    movel([0.098799, -1.267292, -2.641925, -0.803171, 1.570796, 1.669595],accel_mss,speed_ms,0,blend_radius_m)
    movel([0.098967, -1.267010, -2.642082, -0.803297, 1.570796, 1.669764],accel_mss,speed_ms,0,blend_radius_m)
    movel([0.099464, -1.266678, -2.642266, -0.803445, 1.570796, 1.670261],accel_mss,speed_ms,0,blend_radius_m)
    speed_ms = 0.003
    movel([0.099464, -1.270243, -2.643943, -0.798203, 1.570796, 1.670261],accel_mss,speed_ms,0,blend_radius_m)
    speed_ms = 0.007
    movel([0.099864, -1.269963, -2.644099, -0.798327, 1.570796, 1.670661],accel_mss,speed_ms,0,blend_radius_m)
    movel([0.100140, -1.269497, -2.644358, -0.798534, 1.570796, 1.670936],accel_mss,speed_ms,0,blend_radius_m)
    movel([0.100356, -1.268649, -2.644829, -0.798911, 1.570796, 1.671153],accel_mss,speed_ms,0,blend_radius_m)
    movel([0.100640, -1.266818, -2.645843, -0.799728, 1.570796, 1.671436],accel_mss,speed_ms,0,blend_radius_m)
    movel([0.100880, -1.265181, -2.646746, -0.800463, 1.570796, 1.671677],accel_mss,speed_ms,0,blend_radius_m)
    movel([0.101009, -1.264534, -2.647102, -0.800754, 1.570796, 1.671805],accel_mss,speed_ms,0,blend_radius_m)
    movel([0.101145, -1.264159, -2.647307, -0.800923, 1.570796, 1.671942],accel_mss,speed_ms,0,blend_radius_m)
    movel([0.101358, -1.263870, -2.647466, -0.801053, 1.570796, 1.672154],accel_mss,speed_ms,0,blend_radius_m)
    movel([0.101658, -1.263620, -2.647603, -0.801166, 1.570796, 1.672454],accel_mss,speed_ms,0,blend_radius_m)
    movel([0.102128, -1.263533, -2.647651, -0.801205, 1.570796, 1.672924],accel_mss,speed_ms,0,blend_radius_m)
    movel([0.102340, -1.263694, -2.647563, -0.801132, 1.570796, 1.673136],accel_mss,speed_ms,0,blend_radius_m)
    movel([0.102446, -1.263926, -2.647435, -0.801028, 1.570796, 1.673242],accel_mss,speed_ms,0,blend_radius_m)
    movel([0.102458, -1.264305, -2.647228, -0.800857, 1.570796, 1.673254],accel_mss,speed_ms,0,blend_radius_m)
    movel([0.102379, -1.264992, -2.646850, -0.800548, 1.570796, 1.673176],accel_mss,speed_ms,0,blend_radius_m)
    movel([0.102123, -1.266603, -2.645961, -0.799825, 1.570796, 1.672919],accel_mss,speed_ms,0,blend_radius_m)
    movel([0.101853, -1.268341, -2.645000, -0.799048, 1.570796, 1.672649],accel_mss,speed_ms,0,blend_radius_m)
    movel([0.101798, -1.269088, -2.644586, -0.798716, 1.570796, 1.672594],accel_mss,speed_ms,0,blend_radius_m)
    movel([0.101884, -1.269413, -2.644405, -0.798571, 1.570796, 1.672681],accel_mss,speed_ms,0,blend_radius_m)
    movel([0.102127, -1.269459, -2.644379, -0.798551, 1.570796, 1.672923],accel_mss,speed_ms,0,blend_radius_m)
    movel([0.102418, -1.269491, -2.644362, -0.798537, 1.570796, 1.673214],accel_mss,speed_ms,0,blend_radius_m)
    movel([0.102637, -1.269624, -2.644288, -0.798478, 1.570796, 1.673433],accel_mss,speed_ms,0,blend_radius_m)
    movel([0.102685, -1.269900, -2.644134, -0.798355, 1.570796, 1.673481],accel_mss,speed_ms,0,blend_radius_m)
    movel([0.102479, -1.270544, -2.643776, -0.798070, 1.570796, 1.673275],accel_mss,speed_ms,0,blend_radius_m)
    movel([0.102314, -1.270823, -2.643620, -0.797946, 1.570796, 1.673111],accel_mss,speed_ms,0,blend_radius_m)
    movel([0.101871, -1.271146, -2.643440, -0.797803, 1.570796, 1.672667],accel_mss,speed_ms,0,blend_radius_m)
    movel([0.101580, -1.271362, -2.643319, -0.797707, 1.570796, 1.672376],accel_mss,speed_ms,0,blend_radius_m)
    movel([0.101261, -1.271773, -2.643090, -0.797526, 1.570796, 1.672057],accel_mss,speed_ms,0,blend_radius_m)
    movel([0.100848, -1.272313, -2.642788, -0.797288, 1.570796, 1.671644],accel_mss,speed_ms,0,blend_radius_m)
    movel([0.100469, -1.272559, -2.642650, -0.797179, 1.570796, 1.671265],accel_mss,speed_ms,0,blend_radius_m)
    movel([0.100136, -1.272520, -2.642672, -0.797197, 1.570796, 1.670932],accel_mss,speed_ms,0,blend_radius_m)
    movel([0.099864, -1.272178, -2.642863, -0.797347, 1.570796, 1.670660],accel_mss,speed_ms,0,blend_radius_m)
    movel([0.099641, -1.271932, -2.643001, -0.797456, 1.570796, 1.670438],accel_mss,speed_ms,0,blend_radius_m)
    movel([0.099334, -1.271905, -2.643016, -0.797468, 1.570796, 1.670130],accel_mss,speed_ms,0,blend_radius_m)
    movel([0.098951, -1.271937, -2.642998, -0.797454, 1.570796, 1.669747],accel_mss,speed_ms,0,blend_radius_m)
    movel([0.098703, -1.271840, -2.643053, -0.797497, 1.570796, 1.669500],accel_mss,speed_ms,0,blend_radius_m)
    movel([0.098605, -1.271610, -2.643181, -0.797598, 1.570796, 1.669401],accel_mss,speed_ms,0,blend_radius_m)
    movel([0.098652, -1.271263, -2.643375, -0.797751, 1.570796, 1.669448],accel_mss,speed_ms,0,blend_radius_m)
    movel([0.098799, -1.270856, -2.643602, -0.797931, 1.570796, 1.669595],accel_mss,speed_ms,0,blend_radius_m)
    movel([0.098967, -1.270575, -2.643758, -0.798056, 1.570796, 1.669764],accel_mss,speed_ms,0,blend_radius_m)
    movel([0.099464, -1.270243, -2.643943, -0.798203, 1.570796, 1.670261],accel_mss,speed_ms,0,blend_radius_m)
    speed_ms = 0.003
    movel([0.099464, -1.256163, -2.637185, -0.819041, 1.570796, 1.670261],accel_mss,speed_ms,0,blend_radius_m)
    speed_ms = 1.000
    movel([0.099464, -1.229425, -2.623288, -0.859676, 1.570796, 1.670261],accel_mss,speed_ms,0,blend_radius_m)
    movel([0.085805, -1.233581, -2.621092, -0.857716, 1.570796, 1.656601],accel_mss,speed_ms,0,blend_radius_m)
    movel([0.085805, -1.260270, -2.634934, -0.817185, 1.570796, 1.656601],accel_mss,speed_ms,0,blend_radius_m)
    speed_ms = 0.003
    movel([0.085805, -1.270762, -2.639994, -0.801634, 1.570796, 1.656601],accel_mss,speed_ms,0,blend_radius_m)
    speed_ms = 0.007
    movel([0.086070, -1.265880, -2.642708, -0.803802, 1.570796, 1.656867],accel_mss,speed_ms,0,blend_radius_m)
    movel([0.086295, -1.263990, -2.643750, -0.804649, 1.570796, 1.657092],accel_mss,speed_ms,0,blend_radius_m)
    movel([0.086599, -1.262035, -2.644825, -0.805530, 1.570796, 1.657396],accel_mss,speed_ms,0,blend_radius_m)
    movel([0.086929, -1.260286, -2.645781, -0.806321, 1.570796, 1.657725],accel_mss,speed_ms,0,blend_radius_m)
    movel([0.087180, -1.259543, -2.646187, -0.806659, 1.570796, 1.657976],accel_mss,speed_ms,0,blend_radius_m)
    movel([0.087885, -1.258813, -2.646585, -0.806992, 1.570796, 1.658681],accel_mss,speed_ms,0,blend_radius_m)
    movel([0.089726, -1.257950, -2.647054, -0.807385, 1.570796, 1.660522],accel_mss,speed_ms,0,blend_radius_m)
    movel([0.092956, -1.256741, -2.647709, -0.807938, 1.570796, 1.663752],accel_mss,speed_ms,0,blend_radius_m)
    movel([0.099627, -1.254504, -2.648919, -0.808966, 1.570796, 1.670423],accel_mss,speed_ms,0,blend_radius_m)
    movel([0.109598, -1.251283, -2.650649, -0.810457, 1.570796, 1.680394],accel_mss,speed_ms,0,blend_radius_m)
    movel([0.114228, -1.249893, -2.651392, -0.811104, 1.570796, 1.685025],accel_mss,speed_ms,0,blend_radius_m)
    movel([0.116925, -1.249198, -2.651762, -0.811429, 1.570796, 1.687721],accel_mss,speed_ms,0,blend_radius_m)
    movel([0.117802, -1.249298, -2.651709, -0.811382, 1.570796, 1.688598],accel_mss,speed_ms,0,blend_radius_m)
    movel([0.118115, -1.249499, -2.651602, -0.811289, 1.570796, 1.688912],accel_mss,speed_ms,0,blend_radius_m)
    movel([0.117518, -1.253510, -2.649454, -0.809425, 1.570796, 1.688314],accel_mss,speed_ms,0,blend_radius_m)
    movel([0.117200, -1.255550, -2.648354, -0.808485, 1.570796, 1.687996],accel_mss,speed_ms,0,blend_radius_m)
    movel([0.116930, -1.257094, -2.647518, -0.807777, 1.570796, 1.687727],accel_mss,speed_ms,0,blend_radius_m)
    movel([0.116660, -1.258388, -2.646816, -0.807185, 1.570796, 1.687457],accel_mss,speed_ms,0,blend_radius_m)
    movel([0.116358, -1.259620, -2.646145, -0.806624, 1.570796, 1.687154],accel_mss,speed_ms,0,blend_radius_m)
    movel([0.115266, -1.263334, -2.644111, -0.804944, 1.570796, 1.686062],accel_mss,speed_ms,0,blend_radius_m)
    movel([0.114094, -1.266630, -2.642293, -0.803466, 1.570796, 1.684890],accel_mss,speed_ms,0,blend_radius_m)
    movel([0.112789, -1.269640, -2.640620, -0.802129, 1.570796, 1.683586],accel_mss,speed_ms,0,blend_radius_m)
    movel([0.111308, -1.272482, -2.639030, -0.800877, 1.570796, 1.682104],accel_mss,speed_ms,0,blend_radius_m)
    movel([0.109151, -1.275877, -2.637118, -0.799394, 1.570796, 1.679948],accel_mss,speed_ms,0,blend_radius_m)
    movel([0.106892, -1.278659, -2.635541, -0.798189, 1.570796, 1.677688],accel_mss,speed_ms,0,blend_radius_m)
    movel([0.104397, -1.280981, -2.634217, -0.797191, 1.570796, 1.675193],accel_mss,speed_ms,0,blend_radius_m)
    movel([0.101531, -1.282996, -2.633062, -0.796331, 1.570796, 1.672327],accel_mss,speed_ms,0,blend_radius_m)
    movel([0.100843, -1.283390, -2.632836, -0.796163, 1.570796, 1.671639],accel_mss,speed_ms,0,blend_radius_m)
    movel([0.100214, -1.283699, -2.632658, -0.796032, 1.570796, 1.671010],accel_mss,speed_ms,0,blend_radius_m)
    movel([0.099441, -1.284018, -2.632475, -0.795896, 1.570796, 1.670237],accel_mss,speed_ms,0,blend_radius_m)
    movel([0.098221, -1.284469, -2.632215, -0.795705, 1.570796, 1.669018],accel_mss,speed_ms,0,blend_radius_m)
    movel([0.096957, -1.284915, -2.631958, -0.795516, 1.570796, 1.667754],accel_mss,speed_ms,0,blend_radius_m)
    movel([0.096211, -1.285147, -2.631824, -0.795418, 1.570796, 1.667007],accel_mss,speed_ms,0,blend_radius_m)
    movel([0.095602, -1.285283, -2.631746, -0.795360, 1.570796, 1.666399],accel_mss,speed_ms,0,blend_radius_m)
    movel([0.094884, -1.285382, -2.631688, -0.795318, 1.570796, 1.665680],accel_mss,speed_ms,0,blend_radius_m)
    movel([0.092619, -1.285335, -2.631716, -0.795338, 1.570796, 1.663416],accel_mss,speed_ms,0,blend_radius_m)
    movel([0.090657, -1.284691, -2.632087, -0.795611, 1.570796, 1.661453],accel_mss,speed_ms,0,blend_radius_m)
    movel([0.089028, -1.283443, -2.632805, -0.796140, 1.570796, 1.659824],accel_mss,speed_ms,0,blend_radius_m)
    movel([0.087745, -1.281605, -2.633860, -0.796924, 1.570796, 1.658541],accel_mss,speed_ms,0,blend_radius_m)
    movel([0.086658, -1.278724, -2.635504, -0.798161, 1.570796, 1.657455],accel_mss,speed_ms,0,blend_radius_m)
    movel([0.086008, -1.275074, -2.637572, -0.799743, 1.570796, 1.656804],accel_mss,speed_ms,0,blend_radius_m)
    movel([0.085805, -1.270762, -2.639994, -0.801634, 1.570796, 1.656601],accel_mss,speed_ms,0,blend_radius_m)
    speed_ms = 0.003
    movel([0.085805, -1.274319, -2.641664, -0.796406, 1.570796, 1.656601],accel_mss,speed_ms,0,blend_radius_m)
    speed_ms = 0.007
    movel([0.086070, -1.269446, -2.644386, -0.798556, 1.570796, 1.656867],accel_mss,speed_ms,0,blend_radius_m)
    movel([0.086295, -1.267560, -2.645432, -0.799396, 1.570796, 1.657092],accel_mss,speed_ms,0,blend_radius_m)
    movel([0.086599, -1.265609, -2.646510, -0.800270, 1.570796, 1.657396],accel_mss,speed_ms,0,blend_radius_m)
    movel([0.086929, -1.263864, -2.647469, -0.801056, 1.570796, 1.657725],accel_mss,speed_ms,0,blend_radius_m)
    movel([0.087180, -1.263122, -2.647876, -0.801391, 1.570796, 1.657976],accel_mss,speed_ms,0,blend_radius_m)
    movel([0.087885, -1.262393, -2.648275, -0.801720, 1.570796, 1.658681],accel_mss,speed_ms,0,blend_radius_m)
    movel([0.089726, -1.261532, -2.648746, -0.802111, 1.570796, 1.660522],accel_mss,speed_ms,0,blend_radius_m)
    movel([0.092956, -1.260326, -2.649404, -0.802659, 1.570796, 1.663752],accel_mss,speed_ms,0,blend_radius_m)
    movel([0.099627, -1.258093, -2.650617, -0.803680, 1.570796, 1.670423],accel_mss,speed_ms,0,blend_radius_m)
    movel([0.109598, -1.254878, -2.652352, -0.805159, 1.570796, 1.680394],accel_mss,speed_ms,0,blend_radius_m)
    movel([0.114228, -1.253491, -2.653097, -0.805801, 1.570796, 1.685025],accel_mss,speed_ms,0,blend_radius_m)
    movel([0.116925, -1.252797, -2.653469, -0.806123, 1.570796, 1.687721],accel_mss,speed_ms,0,blend_radius_m)
    movel([0.117802, -1.252896, -2.653416, -0.806077, 1.570796, 1.688598],accel_mss,speed_ms,0,blend_radius_m)
    movel([0.118115, -1.253097, -2.653308, -0.805984, 1.570796, 1.688912],accel_mss,speed_ms,0,blend_radius_m)
    movel([0.117518, -1.257101, -2.651153, -0.804135, 1.570796, 1.688314],accel_mss,speed_ms,0,blend_radius_m)
    movel([0.117200, -1.259137, -2.650050, -0.803202, 1.570796, 1.687996],accel_mss,speed_ms,0,blend_radius_m)
    movel([0.116930, -1.260678, -2.649212, -0.802499, 1.570796, 1.687727],accel_mss,speed_ms,0,blend_radius_m)
    movel([0.116660, -1.261969, -2.648507, -0.801913, 1.570796, 1.687457],accel_mss,speed_ms,0,blend_radius_m)
    movel([0.116358, -1.263199, -2.647834, -0.801356, 1.570796, 1.687154],accel_mss,speed_ms,0,blend_radius_m)
    movel([0.115266, -1.266906, -2.645794, -0.799689, 1.570796, 1.686062],accel_mss,speed_ms,0,blend_radius_m)
    movel([0.114094, -1.270195, -2.643970, -0.798224, 1.570796, 1.684890],accel_mss,speed_ms,0,blend_radius_m)
    movel([0.112789, -1.273199, -2.642292, -0.796898, 1.570796, 1.683586],accel_mss,speed_ms,0,blend_radius_m)
    movel([0.111308, -1.276036, -2.640697, -0.795656, 1.570796, 1.682104],accel_mss,speed_ms,0,blend_radius_m)
    movel([0.109151, -1.279423, -2.638780, -0.794186, 1.570796, 1.679948],accel_mss,speed_ms,0,blend_radius_m)
    movel([0.106892, -1.282199, -2.637198, -0.792992, 1.570796, 1.677688],accel_mss,speed_ms,0,blend_radius_m)
    movel([0.104397, -1.284517, -2.635870, -0.792003, 1.570796, 1.675193],accel_mss,speed_ms,0,blend_radius_m)
    movel([0.101531, -1.286527, -2.634712, -0.791150, 1.570796, 1.672327],accel_mss,speed_ms,0,blend_radius_m)
    movel([0.100843, -1.286920, -2.634485, -0.790984, 1.570796, 1.671639],accel_mss,speed_ms,0,blend_radius_m)
    movel([0.100214, -1.287229, -2.634306, -0.790853, 1.570796, 1.671010],accel_mss,speed_ms,0,blend_radius_m)
    movel([0.099441, -1.287548, -2.634122, -0.790719, 1.570796, 1.670237],accel_mss,speed_ms,0,blend_radius_m)
    movel([0.098221, -1.287998, -2.633862, -0.790530, 1.570796, 1.669018],accel_mss,speed_ms,0,blend_radius_m)
    movel([0.096957, -1.288442, -2.633604, -0.790343, 1.570796, 1.667754],accel_mss,speed_ms,0,blend_radius_m)
    movel([0.096211, -1.288674, -2.633470, -0.790245, 1.570796, 1.667007],accel_mss,speed_ms,0,blend_radius_m)
    movel([0.095602, -1.288810, -2.633391, -0.790188, 1.570796, 1.666399],accel_mss,speed_ms,0,blend_radius_m)
    movel([0.094884, -1.288909, -2.633334, -0.790147, 1.570796, 1.665680],accel_mss,speed_ms,0,blend_radius_m)
    movel([0.092619, -1.288862, -2.633361, -0.790166, 1.570796, 1.663416],accel_mss,speed_ms,0,blend_radius_m)
    movel([0.090657, -1.288219, -2.633734, -0.790437, 1.570796, 1.661453],accel_mss,speed_ms,0,blend_radius_m)
    movel([0.089028, -1.286974, -2.634454, -0.790961, 1.570796, 1.659824],accel_mss,speed_ms,0,blend_radius_m)
    movel([0.087745, -1.285140, -2.635511, -0.791738, 1.570796, 1.658541],accel_mss,speed_ms,0,blend_radius_m)
    movel([0.086658, -1.282264, -2.637161, -0.792964, 1.570796, 1.657455],accel_mss,speed_ms,0,blend_radius_m)
    movel([0.086008, -1.278622, -2.639235, -0.794532, 1.570796, 1.656804],accel_mss,speed_ms,0,blend_radius_m)
    movel([0.085805, -1.274319, -2.641664, -0.796406, 1.570796, 1.656601],accel_mss,speed_ms,0,blend_radius_m)
    speed_ms = 0.003
    movel([0.085805, -1.260270, -2.634934, -0.817185, 1.570796, 1.656601],accel_mss,speed_ms,0,blend_radius_m)
    speed_ms = 1.000
    movel([0.085805, -1.233581, -2.621092, -0.857716, 1.570796, 1.656601],accel_mss,speed_ms,0,blend_radius_m)
    movel([0.090276, -1.249111, -2.612707, -0.850572, 1.570796, 1.661072],accel_mss,speed_ms,0,blend_radius_m)
    movel([0.090276, -1.275607, -2.626344, -0.810438, 1.570796, 1.661072],accel_mss,speed_ms,0,blend_radius_m)
    speed_ms = 0.003
    movel([0.090276, -1.286010, -2.631326, -0.795053, 1.570796, 1.661072],accel_mss,speed_ms,0,blend_radius_m)
    speed_ms = 0.007
    speed_ms = 0.003
    movel([0.090276, -1.289535, -2.632970, -0.789884, 1.570796, 1.661072],accel_mss,speed_ms,0,blend_radius_m)
    speed_ms = 0.007
    speed_ms = 0.003
    movel([0.090276, -1.275607, -2.626344, -0.810438, 1.570796, 1.661072],accel_mss,speed_ms,0,blend_radius_m)
    speed_ms = 1.000
    movel([0.090276, -1.249111, -2.612707, -0.850572, 1.570796, 1.661072],accel_mss,speed_ms,0,blend_radius_m)
    movel([0.090517, -1.275491, -2.626410, -0.810488, 1.570796, 1.661314],accel_mss,speed_ms,0,blend_radius_m)
    speed_ms = 0.003
    movel([0.090517, -1.285894, -2.631393, -0.795102, 1.570796, 1.661314],accel_mss,speed_ms,0,blend_radius_m)
    speed_ms = 0.007
    movel([0.090760, -1.285956, -2.631357, -0.795076, 1.570796, 1.661556],accel_mss,speed_ms,0,blend_radius_m)
    movel([0.091359, -1.285967, -2.631351, -0.795071, 1.570796, 1.662155],accel_mss,speed_ms,0,blend_radius_m)
    movel([0.091835, -1.286012, -2.631325, -0.795052, 1.570796, 1.662631],accel_mss,speed_ms,0,blend_radius_m)
    movel([0.092380, -1.286070, -2.631291, -0.795028, 1.570796, 1.663177],accel_mss,speed_ms,0,blend_radius_m)
    movel([0.092996, -1.286119, -2.631263, -0.795007, 1.570796, 1.663793],accel_mss,speed_ms,0,blend_radius_m)
    movel([0.093656, -1.286137, -2.631252, -0.795000, 1.570796, 1.664452],accel_mss,speed_ms,0,blend_radius_m)
    movel([0.094270, -1.286128, -2.631258, -0.795004, 1.570796, 1.665066],accel_mss,speed_ms,0,blend_radius_m)
    movel([0.094742, -1.286082, -2.631284, -0.795023, 1.570796, 1.665538],accel_mss,speed_ms,0,blend_radius_m)
    movel([0.097078, -1.285558, -2.631587, -0.795244, 1.570796, 1.667875],accel_mss,speed_ms,0,blend_radius_m)
    movel([0.099439, -1.284682, -2.632092, -0.795615, 1.570796, 1.670236],accel_mss,speed_ms,0,blend_radius_m)
    movel([0.101784, -1.283471, -2.632789, -0.796129, 1.570796, 1.672581],accel_mss,speed_ms,0,blend_radius_m)
    movel([0.104076, -1.281941, -2.633667, -0.796780, 1.570796, 1.674873],accel_mss,speed_ms,0,blend_radius_m)
    movel([0.104777, -1.281474, -2.633935, -0.796980, 1.570796, 1.675573],accel_mss,speed_ms,0,blend_radius_m)
    movel([0.105551, -1.281055, -2.634174, -0.797159, 1.570796, 1.676347],accel_mss,speed_ms,0,blend_radius_m)
    movel([0.106203, -1.280776, -2.634334, -0.797279, 1.570796, 1.676999],accel_mss,speed_ms,0,blend_radius_m)
    movel([0.106394, -1.280924, -2.634249, -0.797216, 1.570796, 1.677190],accel_mss,speed_ms,0,blend_radius_m)
    movel([0.106666, -1.280931, -2.634245, -0.797212, 1.570796, 1.677462],accel_mss,speed_ms,0,blend_radius_m)
    movel([0.106922, -1.280639, -2.634412, -0.797338, 1.570796, 1.677719],accel_mss,speed_ms,0,blend_radius_m)
    movel([0.107235, -1.280554, -2.634461, -0.797374, 1.570796, 1.678032],accel_mss,speed_ms,0,blend_radius_m)
    movel([0.106944, -1.280659, -2.634401, -0.797329, 1.570796, 1.677741],accel_mss,speed_ms,0,blend_radius_m)
    movel([0.107092, -1.280910, -2.634257, -0.797222, 1.570796, 1.677889],accel_mss,speed_ms,0,blend_radius_m)
    movel([0.107397, -1.280825, -2.634306, -0.797258, 1.570796, 1.678194],accel_mss,speed_ms,0,blend_radius_m)
    movel([0.107675, -1.280853, -2.634290, -0.797246, 1.570796, 1.678471],accel_mss,speed_ms,0,blend_radius_m)
    movel([0.107807, -1.281013, -2.634199, -0.797178, 1.570796, 1.678603],accel_mss,speed_ms,0,blend_radius_m)
    movel([0.108113, -1.280823, -2.634307, -0.797259, 1.570796, 1.678910],accel_mss,speed_ms,0,blend_radius_m)
    movel([0.107859, -1.280759, -2.634344, -0.797287, 1.570796, 1.678655],accel_mss,speed_ms,0,blend_radius_m)
    movel([0.107530, -1.280639, -2.634412, -0.797338, 1.570796, 1.678327],accel_mss,speed_ms,0,blend_radius_m)
    movel([0.108087, -1.280418, -2.634538, -0.797433, 1.570796, 1.678883],accel_mss,speed_ms,0,blend_radius_m)
    movel([0.108555, -1.280456, -2.634517, -0.797416, 1.570796, 1.679351],accel_mss,speed_ms,0,blend_radius_m)
    movel([0.109052, -1.280655, -2.634403, -0.797331, 1.570796, 1.679849],accel_mss,speed_ms,0,blend_radius_m)
    movel([0.109447, -1.280935, -2.634243, -0.797211, 1.570796, 1.680244],accel_mss,speed_ms,0,blend_radius_m)
    movel([0.109568, -1.281224, -2.634078, -0.797087, 1.570796, 1.680365],accel_mss,speed_ms,0,blend_radius_m)
    movel([0.109559, -1.281633, -2.633843, -0.796912, 1.570796, 1.680355],accel_mss,speed_ms,0,blend_radius_m)
    movel([0.109485, -1.281925, -2.633676, -0.796787, 1.570796, 1.680281],accel_mss,speed_ms,0,blend_radius_m)
    movel([0.109326, -1.282211, -2.633512, -0.796665, 1.570796, 1.680122],accel_mss,speed_ms,0,blend_radius_m)
    movel([0.109017, -1.282599, -2.633290, -0.796500, 1.570796, 1.679813],accel_mss,speed_ms,0,blend_radius_m)
    movel([0.108778, -1.282857, -2.633142, -0.796390, 1.570796, 1.679574],accel_mss,speed_ms,0,blend_radius_m)
    movel([0.108466, -1.283158, -2.632969, -0.796262, 1.570796, 1.679263],accel_mss,speed_ms,0,blend_radius_m)
    movel([0.108137, -1.283451, -2.632801, -0.796137, 1.570796, 1.678934],accel_mss,speed_ms,0,blend_radius_m)
    movel([0.107842, -1.283689, -2.632664, -0.796036, 1.570796, 1.678638],accel_mss,speed_ms,0,blend_radius_m)
    movel([0.107121, -1.284217, -2.632360, -0.795812, 1.570796, 1.677917],accel_mss,speed_ms,0,blend_radius_m)
    movel([0.106892, -1.284128, -2.632412, -0.795850, 1.570796, 1.677688],accel_mss,speed_ms,0,blend_radius_m)
    movel([0.107390, -1.283544, -2.632747, -0.796097, 1.570796, 1.678187],accel_mss,speed_ms,0,blend_radius_m)
    movel([0.107724, -1.283168, -2.632963, -0.796257, 1.570796, 1.678521],accel_mss,speed_ms,0,blend_radius_m)
    movel([0.107352, -1.283374, -2.632845, -0.796170, 1.570796, 1.678148],accel_mss,speed_ms,0,blend_radius_m)
    movel([0.107190, -1.283667, -2.632676, -0.796045, 1.570796, 1.677986],accel_mss,speed_ms,0,blend_radius_m)
    movel([0.106820, -1.283786, -2.632609, -0.795995, 1.570796, 1.677616],accel_mss,speed_ms,0,blend_radius_m)
    movel([0.106429, -1.284151, -2.632398, -0.795840, 1.570796, 1.677225],accel_mss,speed_ms,0,blend_radius_m)
    movel([0.106409, -1.284430, -2.632238, -0.795722, 1.570796, 1.677205],accel_mss,speed_ms,0,blend_radius_m)
    movel([0.106162, -1.284337, -2.632291, -0.795761, 1.570796, 1.676958],accel_mss,speed_ms,0,blend_radius_m)
    movel([0.105915, -1.284689, -2.632088, -0.795612, 1.570796, 1.676711],accel_mss,speed_ms,0,blend_radius_m)
    movel([0.106042, -1.284980, -2.631921, -0.795489, 1.570796, 1.676838],accel_mss,speed_ms,0,blend_radius_m)
    movel([0.106016, -1.285267, -2.631755, -0.795367, 1.570796, 1.676812],accel_mss,speed_ms,0,blend_radius_m)
    movel([0.106280, -1.285257, -2.631760, -0.795371, 1.570796, 1.677077],accel_mss,speed_ms,0,blend_radius_m)
    movel([0.106205, -1.285570, -2.631580, -0.795239, 1.570796, 1.677002],accel_mss,speed_ms,0,blend_radius_m)
    movel([0.106244, -1.285829, -2.631431, -0.795130, 1.570796, 1.677041],accel_mss,speed_ms,0,blend_radius_m)
    movel([0.106515, -1.285998, -2.631333, -0.795058, 1.570796, 1.677311],accel_mss,speed_ms,0,blend_radius_m)
    movel([0.106800, -1.285814, -2.631439, -0.795136, 1.570796, 1.677596],accel_mss,speed_ms,0,blend_radius_m)
    movel([0.106483, -1.285854, -2.631416, -0.795119, 1.570796, 1.677280],accel_mss,speed_ms,0,blend_radius_m)
    movel([0.106363, -1.285576, -2.631576, -0.795236, 1.570796, 1.677160],accel_mss,speed_ms,0,blend_radius_m)
    movel([0.106782, -1.285404, -2.631676, -0.795309, 1.570796, 1.677578],accel_mss,speed_ms,0,blend_radius_m)
    movel([0.106980, -1.285541, -2.631597, -0.795251, 1.570796, 1.677777],accel_mss,speed_ms,0,blend_radius_m)
    movel([0.107145, -1.285783, -2.631457, -0.795149, 1.570796, 1.677941],accel_mss,speed_ms,0,blend_radius_m)
    movel([0.107185, -1.286078, -2.631287, -0.795025, 1.570796, 1.677981],accel_mss,speed_ms,0,blend_radius_m)
    movel([0.107094, -1.286383, -2.631110, -0.794896, 1.570796, 1.677891],accel_mss,speed_ms,0,blend_radius_m)
    movel([0.106889, -1.286660, -2.630950, -0.794779, 1.570796, 1.677685],accel_mss,speed_ms,0,blend_radius_m)
    movel([0.106730, -1.287021, -2.630741, -0.794627, 1.570796, 1.677527],accel_mss,speed_ms,0,blend_radius_m)
    movel([0.106361, -1.287438, -2.630499, -0.794452, 1.570796, 1.677157],accel_mss,speed_ms,0,blend_radius_m)
    movel([0.106023, -1.287751, -2.630318, -0.794321, 1.570796, 1.676819],accel_mss,speed_ms,0,blend_radius_m)
    movel([0.105735, -1.287964, -2.630194, -0.794231, 1.570796, 1.676531],accel_mss,speed_ms,0,blend_radius_m)
    movel([0.105337, -1.288150, -2.630086, -0.794153, 1.570796, 1.676133],accel_mss,speed_ms,0,blend_radius_m)
    movel([0.104955, -1.288387, -2.629948, -0.794054, 1.570796, 1.675752],accel_mss,speed_ms,0,blend_radius_m)
    movel([0.104548, -1.288586, -2.629833, -0.793970, 1.570796, 1.675345],accel_mss,speed_ms,0,blend_radius_m)
    movel([0.103748, -1.288777, -2.629722, -0.793890, 1.570796, 1.674544],accel_mss,speed_ms,0,blend_radius_m)
    movel([0.103011, -1.289005, -2.629589, -0.793795, 1.570796, 1.673807],accel_mss,speed_ms,0,blend_radius_m)
    movel([0.102355, -1.289248, -2.629448, -0.793694, 1.570796, 1.673152],accel_mss,speed_ms,0,blend_radius_m)
    movel([0.101965, -1.289540, -2.629278, -0.793572, 1.570796, 1.672761],accel_mss,speed_ms,0,blend_radius_m)
    movel([0.101499, -1.289699, -2.629185, -0.793505, 1.570796, 1.672295],accel_mss,speed_ms,0,blend_radius_m)
    movel([0.101150, -1.289866, -2.629088, -0.793435, 1.570796, 1.671947],accel_mss,speed_ms,0,blend_radius_m)
    movel([0.100675, -1.289847, -2.629098, -0.793443, 1.570796, 1.671471],accel_mss,speed_ms,0,blend_radius_m)
    movel([0.100391, -1.289890, -2.629073, -0.793425, 1.570796, 1.671188],accel_mss,speed_ms,0,blend_radius_m)
    movel([0.100053, -1.290183, -2.628903, -0.793303, 1.570796, 1.670849],accel_mss,speed_ms,0,blend_radius_m)
    movel([0.100321, -1.290199, -2.628893, -0.793297, 1.570796, 1.671118],accel_mss,speed_ms,0,blend_radius_m)
    movel([0.100651, -1.290151, -2.628921, -0.793317, 1.570796, 1.671448],accel_mss,speed_ms,0,blend_radius_m)
    movel([0.101031, -1.290134, -2.628931, -0.793324, 1.570796, 1.671827],accel_mss,speed_ms,0,blend_radius_m)
    movel([0.101319, -1.290099, -2.628952, -0.793338, 1.570796, 1.672116],accel_mss,speed_ms,0,blend_radius_m)
    movel([0.101619, -1.290054, -2.628978, -0.793357, 1.570796, 1.672416],accel_mss,speed_ms,0,blend_radius_m)
    movel([0.102043, -1.289977, -2.629023, -0.793389, 1.570796, 1.672840],accel_mss,speed_ms,0,blend_radius_m)
    movel([0.101987, -1.289743, -2.629159, -0.793487, 1.570796, 1.672784],accel_mss,speed_ms,0,blend_radius_m)
    movel([0.102373, -1.289772, -2.629142, -0.793475, 1.570796, 1.673169],accel_mss,speed_ms,0,blend_radius_m)
    movel([0.102475, -1.289975, -2.629024, -0.793390, 1.570796, 1.673271],accel_mss,speed_ms,0,blend_radius_m)
    movel([0.102816, -1.289921, -2.629056, -0.793413, 1.570796, 1.673613],accel_mss,speed_ms,0,blend_radius_m)
    movel([0.103104, -1.289884, -2.629077, -0.793428, 1.570796, 1.673901],accel_mss,speed_ms,0,blend_radius_m)
    movel([0.103382, -1.289827, -2.629110, -0.793452, 1.570796, 1.674178],accel_mss,speed_ms,0,blend_radius_m)
    movel([0.103678, -1.289588, -2.629250, -0.793552, 1.570796, 1.674474],accel_mss,speed_ms,0,blend_radius_m)
    movel([0.103359, -1.289746, -2.629157, -0.793485, 1.570796, 1.674155],accel_mss,speed_ms,0,blend_radius_m)
    movel([0.103194, -1.289619, -2.629232, -0.793539, 1.570796, 1.673991],accel_mss,speed_ms,0,blend_radius_m)
    movel([0.103230, -1.289311, -2.629411, -0.793667, 1.570796, 1.674026],accel_mss,speed_ms,0,blend_radius_m)
    movel([0.103561, -1.289000, -2.629592, -0.793797, 1.570796, 1.674358],accel_mss,speed_ms,0,blend_radius_m)
    movel([0.103869, -1.288936, -2.629629, -0.793824, 1.570796, 1.674665],accel_mss,speed_ms,0,blend_radius_m)
    movel([0.103902, -1.289178, -2.629488, -0.793723, 1.570796, 1.674699],accel_mss,speed_ms,0,blend_radius_m)
    movel([0.104086, -1.289372, -2.629376, -0.793642, 1.570796, 1.674882],accel_mss,speed_ms,0,blend_radius_m)
    movel([0.104470, -1.289572, -2.629259, -0.793558, 1.570796, 1.675266],accel_mss,speed_ms,0,blend_radius_m)
    movel([0.104480, -1.289893, -2.629072, -0.793424, 1.570796, 1.675276],accel_mss,speed_ms,0,blend_radius_m)
    movel([0.104166, -1.289990, -2.629015, -0.793384, 1.570796, 1.674962],accel_mss,speed_ms,0,blend_radius_m)
    movel([0.103943, -1.289929, -2.629051, -0.793409, 1.570796, 1.674739],accel_mss,speed_ms,0,blend_radius_m)
    movel([0.103724, -1.289790, -2.629132, -0.793467, 1.570796, 1.674520],accel_mss,speed_ms,0,blend_radius_m)
    movel([0.103804, -1.290067, -2.628970, -0.793352, 1.570796, 1.674600],accel_mss,speed_ms,0,blend_radius_m)
    movel([0.103792, -1.290462, -2.628740, -0.793187, 1.570796, 1.674589],accel_mss,speed_ms,0,blend_radius_m)
    movel([0.103523, -1.290823, -2.628529, -0.793037, 1.570796, 1.674319],accel_mss,speed_ms,0,blend_radius_m)
    movel([0.103297, -1.291104, -2.628365, -0.792920, 1.570796, 1.674094],accel_mss,speed_ms,0,blend_radius_m)
    movel([0.102982, -1.291173, -2.628325, -0.792892, 1.570796, 1.673778],accel_mss,speed_ms,0,blend_radius_m)
    movel([0.102668, -1.291475, -2.628148, -0.792766, 1.570796, 1.673465],accel_mss,speed_ms,0,blend_radius_m)
    movel([0.102281, -1.291681, -2.628027, -0.792680, 1.570796, 1.673077],accel_mss,speed_ms,0,blend_radius_m)
    movel([0.101902, -1.291838, -2.627935, -0.792615, 1.570796, 1.672698],accel_mss,speed_ms,0,blend_radius_m)
    movel([0.101557, -1.291976, -2.627854, -0.792558, 1.570796, 1.672353],accel_mss,speed_ms,0,blend_radius_m)
    movel([0.101243, -1.292105, -2.627779, -0.792505, 1.570796, 1.672039],accel_mss,speed_ms,0,blend_radius_m)
    movel([0.101286, -1.292331, -2.627647, -0.792411, 1.570796, 1.672083],accel_mss,speed_ms,0,blend_radius_m)
    movel([0.100997, -1.292480, -2.627559, -0.792350, 1.570796, 1.671793],accel_mss,speed_ms,0,blend_radius_m)
    movel([0.100718, -1.292440, -2.627583, -0.792366, 1.570796, 1.671514],accel_mss,speed_ms,0,blend_radius_m)
    movel([0.100425, -1.292566, -2.627509, -0.792314, 1.570796, 1.671222],accel_mss,speed_ms,0,blend_radius_m)
    movel([0.099331, -1.293071, -2.627213, -0.792105, 1.570796, 1.670127],accel_mss,speed_ms,0,blend_radius_m)
    movel([0.097242, -1.293784, -2.626794, -0.791811, 1.570796, 1.668038],accel_mss,speed_ms,0,blend_radius_m)
    movel([0.095038, -1.294457, -2.626398, -0.791534, 1.570796, 1.665834],accel_mss,speed_ms,0,blend_radius_m)
    movel([0.093267, -1.294893, -2.626141, -0.791355, 1.570796, 1.664064],accel_mss,speed_ms,0,blend_radius_m)
    movel([0.092796, -1.295002, -2.626077, -0.791310, 1.570796, 1.663592],accel_mss,speed_ms,0,blend_radius_m)
    movel([0.092505, -1.295072, -2.626035, -0.791282, 1.570796, 1.663301],accel_mss,speed_ms,0,blend_radius_m)
    movel([0.092006, -1.295190, -2.625966, -0.791233, 1.570796, 1.662802],accel_mss,speed_ms,0,blend_radius_m)
    movel([0.091686, -1.295204, -2.625958, -0.791227, 1.570796, 1.662483],accel_mss,speed_ms,0,blend_radius_m)
    movel([0.091516, -1.295043, -2.626052, -0.791293, 1.570796, 1.662312],accel_mss,speed_ms,0,blend_radius_m)
    movel([0.090908, -1.295099, -2.626020, -0.791271, 1.570796, 1.661704],accel_mss,speed_ms,0,blend_radius_m)
    movel([0.091012, -1.295287, -2.625909, -0.791193, 1.570796, 1.661808],accel_mss,speed_ms,0,blend_radius_m)
    movel([0.091131, -1.295453, -2.625811, -0.791125, 1.570796, 1.661927],accel_mss,speed_ms,0,blend_radius_m)
    movel([0.091380, -1.295526, -2.625768, -0.791095, 1.570796, 1.662176],accel_mss,speed_ms,0,blend_radius_m)
    movel([0.091703, -1.295529, -2.625766, -0.791094, 1.570796, 1.662500],accel_mss,speed_ms,0,blend_radius_m)
    movel([0.091970, -1.295280, -2.625913, -0.791196, 1.570796, 1.662766],accel_mss,speed_ms,0,blend_radius_m)
    movel([0.092331, -1.295302, -2.625900, -0.791187, 1.570796, 1.663127],accel_mss,speed_ms,0,blend_radius_m)
    movel([0.092659, -1.295213, -2.625953, -0.791224, 1.570796, 1.663455],accel_mss,speed_ms,0,blend_radius_m)
    movel([0.092762, -1.295396, -2.625845, -0.791149, 1.570796, 1.663559],accel_mss,speed_ms,0,blend_radius_m)
    movel([0.092991, -1.295457, -2.625808, -0.791124, 1.570796, 1.663787],accel_mss,speed_ms,0,blend_radius_m)
    movel([0.093296, -1.295278, -2.625914, -0.791197, 1.570796, 1.664092],accel_mss,speed_ms,0,blend_radius_m)
    movel([0.093554, -1.295264, -2.625922, -0.791203, 1.570796, 1.664350],accel_mss,speed_ms,0,blend_radius_m)
    movel([0.093259, -1.295524, -2.625769, -0.791096, 1.570796, 1.664056],accel_mss,speed_ms,0,blend_radius_m)
    movel([0.092956, -1.295608, -2.625719, -0.791062, 1.570796, 1.663753],accel_mss,speed_ms,0,blend_radius_m)
    movel([0.092691, -1.295566, -2.625744, -0.791079, 1.570796, 1.663487],accel_mss,speed_ms,0,blend_radius_m)
    movel([0.092356, -1.295474, -2.625799, -0.791117, 1.570796, 1.663152],accel_mss,speed_ms,0,blend_radius_m)
    movel([0.092063, -1.295519, -2.625772, -0.791098, 1.570796, 1.662859],accel_mss,speed_ms,0,blend_radius_m)
    movel([0.091652, -1.295639, -2.625701, -0.791049, 1.570796, 1.662448],accel_mss,speed_ms,0,blend_radius_m)
    movel([0.091327, -1.295728, -2.625649, -0.791013, 1.570796, 1.662123],accel_mss,speed_ms,0,blend_radius_m)
    movel([0.091035, -1.295784, -2.625615, -0.790989, 1.570796, 1.661832],accel_mss,speed_ms,0,blend_radius_m)
    movel([0.090721, -1.295828, -2.625590, -0.790972, 1.570796, 1.661517],accel_mss,speed_ms,0,blend_radius_m)
    movel([0.090684, -1.295590, -2.625730, -0.791069, 1.570796, 1.661480],accel_mss,speed_ms,0,blend_radius_m)
    movel([0.090510, -1.295461, -2.625806, -0.791122, 1.570796, 1.661306],accel_mss,speed_ms,0,blend_radius_m)
    movel([0.090188, -1.295575, -2.625739, -0.791075, 1.570796, 1.660984],accel_mss,speed_ms,0,blend_radius_m)
    movel([0.090012, -1.295435, -2.625821, -0.791133, 1.570796, 1.660808],accel_mss,speed_ms,0,blend_radius_m)
    movel([0.089943, -1.295224, -2.625946, -0.791219, 1.570796, 1.660739],accel_mss,speed_ms,0,blend_radius_m)
    movel([0.089712, -1.295174, -2.625976, -0.791240, 1.570796, 1.660509],accel_mss,speed_ms,0,blend_radius_m)
    movel([0.089970, -1.294932, -2.626118, -0.791339, 1.570796, 1.660766],accel_mss,speed_ms,0,blend_radius_m)
    movel([0.090285, -1.294888, -2.626144, -0.791357, 1.570796, 1.661081],accel_mss,speed_ms,0,blend_radius_m)
    movel([0.090132, -1.295178, -2.625973, -0.791238, 1.570796, 1.660928],accel_mss,speed_ms,0,blend_radius_m)
    movel([0.090205, -1.295458, -2.625808, -0.791123, 1.570796, 1.661001],accel_mss,speed_ms,0,blend_radius_m)
    movel([0.090261, -1.295173, -2.625976, -0.791240, 1.570796, 1.661057],accel_mss,speed_ms,0,blend_radius_m)
    movel([0.090563, -1.295048, -2.626049, -0.791291, 1.570796, 1.661359],accel_mss,speed_ms,0,blend_radius_m)
    movel([0.090470, -1.294836, -2.626175, -0.791378, 1.570796, 1.661266],accel_mss,speed_ms,0,blend_radius_m)
    movel([0.090383, -1.294562, -2.626336, -0.791491, 1.570796, 1.661179],accel_mss,speed_ms,0,blend_radius_m)
    movel([0.090678, -1.294319, -2.626479, -0.791591, 1.570796, 1.661474],accel_mss,speed_ms,0,blend_radius_m)
    movel([0.090825, -1.293986, -2.626675, -0.791728, 1.570796, 1.661621],accel_mss,speed_ms,0,blend_radius_m)
    movel([0.090518, -1.294183, -2.626559, -0.791647, 1.570796, 1.661314],accel_mss,speed_ms,0,blend_radius_m)
    movel([0.090290, -1.294420, -2.626420, -0.791549, 1.570796, 1.661086],accel_mss,speed_ms,0,blend_radius_m)
    movel([0.090113, -1.294706, -2.626251, -0.791432, 1.570796, 1.660910],accel_mss,speed_ms,0,blend_radius_m)
    movel([0.089804, -1.294774, -2.626211, -0.791404, 1.570796, 1.660600],accel_mss,speed_ms,0,blend_radius_m)
    movel([0.089954, -1.294457, -2.626398, -0.791534, 1.570796, 1.660750],accel_mss,speed_ms,0,blend_radius_m)
    movel([0.090167, -1.294184, -2.626558, -0.791646, 1.570796, 1.660963],accel_mss,speed_ms,0,blend_radius_m)
    movel([0.090457, -1.293839, -2.626762, -0.791789, 1.570796, 1.661253],accel_mss,speed_ms,0,blend_radius_m)
    movel([0.090350, -1.293548, -2.626933, -0.791909, 1.570796, 1.661146],accel_mss,speed_ms,0,blend_radius_m)
    movel([0.090002, -1.293462, -2.626983, -0.791944, 1.570796, 1.660798],accel_mss,speed_ms,0,blend_radius_m)
    movel([0.089628, -1.293427, -2.627004, -0.791959, 1.570796, 1.660424],accel_mss,speed_ms,0,blend_radius_m)
    movel([0.089304, -1.293469, -2.626979, -0.791941, 1.570796, 1.660101],accel_mss,speed_ms,0,blend_radius_m)
    movel([0.089032, -1.293425, -2.627005, -0.791959, 1.570796, 1.659829],accel_mss,speed_ms,0,blend_radius_m)
    movel([0.088749, -1.293465, -2.626981, -0.791943, 1.570796, 1.659546],accel_mss,speed_ms,0,blend_radius_m)
    movel([0.088519, -1.293407, -2.627015, -0.791966, 1.570796, 1.659315],accel_mss,speed_ms,0,blend_radius_m)
    movel([0.088260, -1.293283, -2.627088, -0.792018, 1.570796, 1.659057],accel_mss,speed_ms,0,blend_radius_m)
    movel([0.087984, -1.293094, -2.627199, -0.792096, 1.570796, 1.658780],accel_mss,speed_ms,0,blend_radius_m)
    movel([0.087838, -1.292892, -2.627318, -0.792179, 1.570796, 1.658634],accel_mss,speed_ms,0,blend_radius_m)
    movel([0.087930, -1.292619, -2.627478, -0.792292, 1.570796, 1.658726],accel_mss,speed_ms,0,blend_radius_m)
    movel([0.088018, -1.292324, -2.627651, -0.792414, 1.570796, 1.658814],accel_mss,speed_ms,0,blend_radius_m)
    movel([0.088177, -1.291786, -2.627966, -0.792637, 1.570796, 1.658973],accel_mss,speed_ms,0,blend_radius_m)
    movel([0.088520, -1.291368, -2.628210, -0.792810, 1.570796, 1.659316],accel_mss,speed_ms,0,blend_radius_m)
    movel([0.088850, -1.291076, -2.628381, -0.792932, 1.570796, 1.659647],accel_mss,speed_ms,0,blend_radius_m)
    movel([0.089096, -1.290851, -2.628513, -0.793025, 1.570796, 1.659893],accel_mss,speed_ms,0,blend_radius_m)
    movel([0.089150, -1.290478, -2.628730, -0.793180, 1.570796, 1.659946],accel_mss,speed_ms,0,blend_radius_m)
    movel([0.088850, -1.290441, -2.628752, -0.793196, 1.570796, 1.659646],accel_mss,speed_ms,0,blend_radius_m)
    movel([0.088651, -1.290304, -2.628832, -0.793253, 1.570796, 1.659447],accel_mss,speed_ms,0,blend_radius_m)
    movel([0.088309, -1.290383, -2.628786, -0.793220, 1.570796, 1.659105],accel_mss,speed_ms,0,blend_radius_m)
    movel([0.087687, -1.290468, -2.628736, -0.793185, 1.570796, 1.658483],accel_mss,speed_ms,0,blend_radius_m)
    movel([0.087026, -1.290337, -2.628813, -0.793239, 1.570796, 1.657823],accel_mss,speed_ms,0,blend_radius_m)
    movel([0.086481, -1.290048, -2.628981, -0.793360, 1.570796, 1.657277],accel_mss,speed_ms,0,blend_radius_m)
    movel([0.086205, -1.289649, -2.629214, -0.793526, 1.570796, 1.657001],accel_mss,speed_ms,0,blend_radius_m)
    movel([0.086167, -1.289347, -2.629390, -0.793652, 1.570796, 1.656963],accel_mss,speed_ms,0,blend_radius_m)
    movel([0.086235, -1.289031, -2.629574, -0.793784, 1.570796, 1.657032],accel_mss,speed_ms,0,blend_radius_m)
    movel([0.086426, -1.288658, -2.629791, -0.793940, 1.570796, 1.657222],accel_mss,speed_ms,0,blend_radius_m)
    movel([0.086757, -1.288197, -2.630059, -0.794133, 1.570796, 1.657553],accel_mss,speed_ms,0,blend_radius_m)
    movel([0.086981, -1.287956, -2.630199, -0.794234, 1.570796, 1.657777],accel_mss,speed_ms,0,blend_radius_m)
    movel([0.087305, -1.287686, -2.630355, -0.794348, 1.570796, 1.658101],accel_mss,speed_ms,0,blend_radius_m)
    movel([0.087627, -1.287459, -2.630487, -0.794443, 1.570796, 1.658423],accel_mss,speed_ms,0,blend_radius_m)
    movel([0.087930, -1.287270, -2.630596, -0.794522, 1.570796, 1.658726],accel_mss,speed_ms,0,blend_radius_m)
    movel([0.088216, -1.287266, -2.630599, -0.794524, 1.570796, 1.659013],accel_mss,speed_ms,0,blend_radius_m)
    movel([0.088406, -1.287400, -2.630521, -0.794468, 1.570796, 1.659202],accel_mss,speed_ms,0,blend_radius_m)
    movel([0.088248, -1.287057, -2.630720, -0.794612, 1.570796, 1.659044],accel_mss,speed_ms,0,blend_radius_m)
    movel([0.088513, -1.286866, -2.630831, -0.794692, 1.570796, 1.659309],accel_mss,speed_ms,0,blend_radius_m)
    movel([0.088853, -1.286547, -2.631015, -0.794827, 1.570796, 1.659650],accel_mss,speed_ms,0,blend_radius_m)
    movel([0.089467, -1.286118, -2.631263, -0.795007, 1.570796, 1.660263],accel_mss,speed_ms,0,blend_radius_m)
    movel([0.090092, -1.285722, -2.631492, -0.795175, 1.570796, 1.660888],accel_mss,speed_ms,0,blend_radius_m)
    movel([0.090426, -1.285649, -2.631534, -0.795205, 1.570796, 1.661223],accel_mss,speed_ms,0,blend_radius_m)
    movel([0.090517, -1.285894, -2.631393, -0.795102, 1.570796, 1.661314],accel_mss,speed_ms,0,blend_radius_m)
    speed_ms = 0.003
    movel([0.090517, -1.289419, -2.633037, -0.789932, 1.570796, 1.661314],accel_mss,speed_ms,0,blend_radius_m)
    speed_ms = 0.007
    movel([0.090760, -1.289481, -2.633001, -0.789907, 1.570796, 1.661556],accel_mss,speed_ms,0,blend_radius_m)
    movel([0.091359, -1.289492, -2.632995, -0.789902, 1.570796, 1.662155],accel_mss,speed_ms,0,blend_radius_m)
    movel([0.091835, -1.289537, -2.632969, -0.789883, 1.570796, 1.662631],accel_mss,speed_ms,0,blend_radius_m)
    movel([0.092380, -1.289595, -2.632935, -0.789859, 1.570796, 1.663177],accel_mss,speed_ms,0,blend_radius_m)
    movel([0.092996, -1.289644, -2.632907, -0.789838, 1.570796, 1.663793],accel_mss,speed_ms,0,blend_radius_m)
    movel([0.093656, -1.289662, -2.632896, -0.789831, 1.570796, 1.664452],accel_mss,speed_ms,0,blend_radius_m)
    movel([0.094270, -1.289652, -2.632902, -0.789835, 1.570796, 1.665066],accel_mss,speed_ms,0,blend_radius_m)
    movel([0.094742, -1.289607, -2.632928, -0.789854, 1.570796, 1.665538],accel_mss,speed_ms,0,blend_radius_m)
    movel([0.097078, -1.289084, -2.633232, -0.790073, 1.570796, 1.667875],accel_mss,speed_ms,0,blend_radius_m)
    movel([0.099439, -1.288210, -2.633739, -0.790440, 1.570796, 1.670236],accel_mss,speed_ms,0,blend_radius_m)
    movel([0.101784, -1.287001, -2.634438, -0.790950, 1.570796, 1.672581],accel_mss,speed_ms,0,blend_radius_m)
    movel([0.104076, -1.285475, -2.635318, -0.791596, 1.570796, 1.674873],accel_mss,speed_ms,0,blend_radius_m)
    movel([0.104777, -1.285009, -2.635587, -0.791794, 1.570796, 1.675573],accel_mss,speed_ms,0,blend_radius_m)
    movel([0.105551, -1.284591, -2.635827, -0.791971, 1.570796, 1.676347],accel_mss,speed_ms,0,blend_radius_m)
    movel([0.106203, -1.284312, -2.635987, -0.792090, 1.570796, 1.676999],accel_mss,speed_ms,0,blend_radius_m)
    movel([0.106394, -1.284460, -2.635902, -0.792027, 1.570796, 1.677190],accel_mss,speed_ms,0,blend_radius_m)
    movel([0.106666, -1.284467, -2.635898, -0.792024, 1.570796, 1.677462],accel_mss,speed_ms,0,blend_radius_m)
    movel([0.106922, -1.284176, -2.636065, -0.792148, 1.570796, 1.677719],accel_mss,speed_ms,0,blend_radius_m)
    movel([0.107235, -1.284090, -2.636114, -0.792184, 1.570796, 1.678032],accel_mss,speed_ms,0,blend_radius_m)
    movel([0.106944, -1.284195, -2.636054, -0.792140, 1.570796, 1.677741],accel_mss,speed_ms,0,blend_radius_m)
    movel([0.107092, -1.284446, -2.635910, -0.792033, 1.570796, 1.677889],accel_mss,speed_ms,0,blend_radius_m)
    movel([0.107397, -1.284361, -2.635959, -0.792069, 1.570796, 1.678194],accel_mss,speed_ms,0,blend_radius_m)
    movel([0.107675, -1.284389, -2.635943, -0.792057, 1.570796, 1.678471],accel_mss,speed_ms,0,blend_radius_m)
    movel([0.107807, -1.284548, -2.635851, -0.791989, 1.570796, 1.678603],accel_mss,speed_ms,0,blend_radius_m)
    movel([0.108113, -1.284359, -2.635960, -0.792070, 1.570796, 1.678910],accel_mss,speed_ms,0,blend_radius_m)
    movel([0.107859, -1.284295, -2.635997, -0.792097, 1.570796, 1.678655],accel_mss,speed_ms,0,blend_radius_m)
    movel([0.107530, -1.284175, -2.636066, -0.792148, 1.570796, 1.678327],accel_mss,speed_ms,0,blend_radius_m)
    movel([0.108087, -1.283955, -2.636192, -0.792242, 1.570796, 1.678883],accel_mss,speed_ms,0,blend_radius_m)
    movel([0.108555, -1.283993, -2.636170, -0.792226, 1.570796, 1.679351],accel_mss,speed_ms,0,blend_radius_m)
    movel([0.109052, -1.284191, -2.636057, -0.792141, 1.570796, 1.679849],accel_mss,speed_ms,0,blend_radius_m)
    movel([0.109447, -1.284471, -2.635896, -0.792022, 1.570796, 1.680244],accel_mss,speed_ms,0,blend_radius_m)
    movel([0.109568, -1.284760, -2.635730, -0.791899, 1.570796, 1.680365],accel_mss,speed_ms,0,blend_radius_m)
    movel([0.109559, -1.285168, -2.635495, -0.791726, 1.570796, 1.680355],accel_mss,speed_ms,0,blend_radius_m)
    movel([0.109485, -1.285459, -2.635327, -0.791602, 1.570796, 1.680281],accel_mss,speed_ms,0,blend_radius_m)
    movel([0.109326, -1.285744, -2.635163, -0.791481, 1.570796, 1.680122],accel_mss,speed_ms,0,blend_radius_m)
    movel([0.109017, -1.286131, -2.634940, -0.791318, 1.570796, 1.679813],accel_mss,speed_ms,0,blend_radius_m)
    movel([0.108778, -1.286389, -2.634792, -0.791209, 1.570796, 1.679574],accel_mss,speed_ms,0,blend_radius_m)
    movel([0.108466, -1.286690, -2.634618, -0.791081, 1.570796, 1.679263],accel_mss,speed_ms,0,blend_radius_m)
    movel([0.108137, -1.286981, -2.634449, -0.790958, 1.570796, 1.678934],accel_mss,speed_ms,0,blend_radius_m)
    movel([0.107842, -1.287219, -2.634312, -0.790858, 1.570796, 1.678638],accel_mss,speed_ms,0,blend_radius_m)
    movel([0.107121, -1.287746, -2.634007, -0.790636, 1.570796, 1.677917],accel_mss,speed_ms,0,blend_radius_m)
    movel([0.106892, -1.287657, -2.634059, -0.790673, 1.570796, 1.677688],accel_mss,speed_ms,0,blend_radius_m)
    movel([0.107390, -1.287075, -2.634396, -0.790919, 1.570796, 1.678187],accel_mss,speed_ms,0,blend_radius_m)
    movel([0.107724, -1.286699, -2.634612, -0.791077, 1.570796, 1.678521],accel_mss,speed_ms,0,blend_radius_m)
    movel([0.107352, -1.286905, -2.634494, -0.790991, 1.570796, 1.678148],accel_mss,speed_ms,0,blend_radius_m)
    movel([0.107190, -1.287198, -2.634325, -0.790867, 1.570796, 1.677986],accel_mss,speed_ms,0,blend_radius_m)
    movel([0.106820, -1.287315, -2.634257, -0.790817, 1.570796, 1.677616],accel_mss,speed_ms,0,blend_radius_m)
    movel([0.106429, -1.287680, -2.634045, -0.790663, 1.570796, 1.677225],accel_mss,speed_ms,0,blend_radius_m)
    movel([0.106409, -1.287958, -2.633885, -0.790546, 1.570796, 1.677205],accel_mss,speed_ms,0,blend_radius_m)
    movel([0.106162, -1.287866, -2.633938, -0.790585, 1.570796, 1.676958],accel_mss,speed_ms,0,blend_radius_m)
    movel([0.105915, -1.288217, -2.633735, -0.790437, 1.570796, 1.676711],accel_mss,speed_ms,0,blend_radius_m)
    movel([0.106042, -1.288507, -2.633567, -0.790315, 1.570796, 1.676838],accel_mss,speed_ms,0,blend_radius_m)
    movel([0.106016, -1.288793, -2.633401, -0.790195, 1.570796, 1.676812],accel_mss,speed_ms,0,blend_radius_m)
    movel([0.106280, -1.288784, -2.633406, -0.790199, 1.570796, 1.677077],accel_mss,speed_ms,0,blend_radius_m)
    movel([0.106205, -1.289096, -2.633225, -0.790068, 1.570796, 1.677002],accel_mss,speed_ms,0,blend_radius_m)
    movel([0.106244, -1.289354, -2.633075, -0.789960, 1.570796, 1.677041],accel_mss,speed_ms,0,blend_radius_m)
    movel([0.106515, -1.289523, -2.632977, -0.789889, 1.570796, 1.677311],accel_mss,speed_ms,0,blend_radius_m)
    movel([0.106800, -1.289339, -2.633084, -0.789966, 1.570796, 1.677596],accel_mss,speed_ms,0,blend_radius_m)
    movel([0.106483, -1.289380, -2.633060, -0.789949, 1.570796, 1.677280],accel_mss,speed_ms,0,blend_radius_m)
    movel([0.106363, -1.289102, -2.633221, -0.790065, 1.570796, 1.677160],accel_mss,speed_ms,0,blend_radius_m)
    movel([0.106782, -1.288931, -2.633321, -0.790137, 1.570796, 1.677578],accel_mss,speed_ms,0,blend_radius_m)
    movel([0.106980, -1.289067, -2.633242, -0.790080, 1.570796, 1.677777],accel_mss,speed_ms,0,blend_radius_m)
    movel([0.107145, -1.289309, -2.633101, -0.789979, 1.570796, 1.677941],accel_mss,speed_ms,0,blend_radius_m)
    movel([0.107185, -1.289603, -2.632931, -0.789856, 1.570796, 1.677981],accel_mss,speed_ms,0,blend_radius_m)
    movel([0.107094, -1.289907, -2.632754, -0.789728, 1.570796, 1.677891],accel_mss,speed_ms,0,blend_radius_m)
    movel([0.106889, -1.290184, -2.632593, -0.789612, 1.570796, 1.677685],accel_mss,speed_ms,0,blend_radius_m)
    movel([0.106730, -1.290544, -2.632383, -0.789462, 1.570796, 1.677527],accel_mss,speed_ms,0,blend_radius_m)
    movel([0.106361, -1.290960, -2.632141, -0.789288, 1.570796, 1.677157],accel_mss,speed_ms,0,blend_radius_m)
    movel([0.106023, -1.291272, -2.631959, -0.789158, 1.570796, 1.676819],accel_mss,speed_ms,0,blend_radius_m)
    movel([0.105735, -1.291485, -2.631835, -0.789069, 1.570796, 1.676531],accel_mss,speed_ms,0,blend_radius_m)
    movel([0.105337, -1.291671, -2.631726, -0.788992, 1.570796, 1.676133],accel_mss,speed_ms,0,blend_radius_m)
    movel([0.104955, -1.291907, -2.631589, -0.788894, 1.570796, 1.675752],accel_mss,speed_ms,0,blend_radius_m)
    movel([0.104548, -1.292105, -2.631472, -0.788811, 1.570796, 1.675345],accel_mss,speed_ms,0,blend_radius_m)
    movel([0.103748, -1.292296, -2.631361, -0.788732, 1.570796, 1.674544],accel_mss,speed_ms,0,blend_radius_m)
    movel([0.103011, -1.292524, -2.631228, -0.788637, 1.570796, 1.673807],accel_mss,speed_ms,0,blend_radius_m)
    movel([0.102355, -1.292766, -2.631086, -0.788537, 1.570796, 1.673152],accel_mss,speed_ms,0,blend_radius_m)
    movel([0.101965, -1.293057, -2.630916, -0.788416, 1.570796, 1.672761],accel_mss,speed_ms,0,blend_radius_m)
    movel([0.101499, -1.293216, -2.630823, -0.788350, 1.570796, 1.672295],accel_mss,speed_ms,0,blend_radius_m)
    movel([0.101150, -1.293383, -2.630725, -0.788281, 1.570796, 1.671947],accel_mss,speed_ms,0,blend_radius_m)
    movel([0.100675, -1.293364, -2.630736, -0.788289, 1.570796, 1.671471],accel_mss,speed_ms,0,blend_radius_m)
    movel([0.100391, -1.293407, -2.630711, -0.788271, 1.570796, 1.671188],accel_mss,speed_ms,0,blend_radius_m)
    movel([0.100053, -1.293699, -2.630540, -0.788150, 1.570796, 1.670849],accel_mss,speed_ms,0,blend_radius_m)
    movel([0.100321, -1.293715, -2.630530, -0.788144, 1.570796, 1.671118],accel_mss,speed_ms,0,blend_radius_m)
    movel([0.100651, -1.293667, -2.630559, -0.788164, 1.570796, 1.671448],accel_mss,speed_ms,0,blend_radius_m)
    movel([0.101031, -1.293650, -2.630569, -0.788171, 1.570796, 1.671827],accel_mss,speed_ms,0,blend_radius_m)
    movel([0.101319, -1.293615, -2.630589, -0.788185, 1.570796, 1.672116],accel_mss,speed_ms,0,blend_radius_m)
    movel([0.101619, -1.293570, -2.630615, -0.788204, 1.570796, 1.672416],accel_mss,speed_ms,0,blend_radius_m)
    movel([0.102043, -1.293494, -2.630660, -0.788235, 1.570796, 1.672840],accel_mss,speed_ms,0,blend_radius_m)
    movel([0.101987, -1.293260, -2.630797, -0.788332, 1.570796, 1.672784],accel_mss,speed_ms,0,blend_radius_m)
    movel([0.102373, -1.293289, -2.630780, -0.788320, 1.570796, 1.673169],accel_mss,speed_ms,0,blend_radius_m)
    movel([0.102475, -1.293491, -2.630662, -0.788236, 1.570796, 1.673271],accel_mss,speed_ms,0,blend_radius_m)
    movel([0.102816, -1.293437, -2.630693, -0.788259, 1.570796, 1.673613],accel_mss,speed_ms,0,blend_radius_m)
    movel([0.103104, -1.293401, -2.630715, -0.788274, 1.570796, 1.673901],accel_mss,speed_ms,0,blend_radius_m)
    movel([0.103382, -1.293344, -2.630748, -0.788297, 1.570796, 1.674178],accel_mss,speed_ms,0,blend_radius_m)
    movel([0.103678, -1.293105, -2.630888, -0.788396, 1.570796, 1.674474],accel_mss,speed_ms,0,blend_radius_m)
    movel([0.103359, -1.293263, -2.630795, -0.788331, 1.570796, 1.674155],accel_mss,speed_ms,0,blend_radius_m)
    movel([0.103194, -1.293136, -2.630870, -0.788383, 1.570796, 1.673991],accel_mss,speed_ms,0,blend_radius_m)
    movel([0.103230, -1.292829, -2.631049, -0.788511, 1.570796, 1.674026],accel_mss,speed_ms,0,blend_radius_m)
    movel([0.103561, -1.292519, -2.631231, -0.788639, 1.570796, 1.674358],accel_mss,speed_ms,0,blend_radius_m)
    movel([0.103869, -1.292455, -2.631268, -0.788666, 1.570796, 1.674665],accel_mss,speed_ms,0,blend_radius_m)
    movel([0.103902, -1.292696, -2.631127, -0.788566, 1.570796, 1.674699],accel_mss,speed_ms,0,blend_radius_m)
    movel([0.104086, -1.292889, -2.631014, -0.788486, 1.570796, 1.674882],accel_mss,speed_ms,0,blend_radius_m)
    movel([0.104470, -1.293089, -2.630897, -0.788403, 1.570796, 1.675266],accel_mss,speed_ms,0,blend_radius_m)
    movel([0.104480, -1.293409, -2.630709, -0.788270, 1.570796, 1.675276],accel_mss,speed_ms,0,blend_radius_m)
    movel([0.104166, -1.293506, -2.630653, -0.788230, 1.570796, 1.674962],accel_mss,speed_ms,0,blend_radius_m)
    movel([0.103943, -1.293445, -2.630688, -0.788255, 1.570796, 1.674739],accel_mss,speed_ms,0,blend_radius_m)
    movel([0.103724, -1.293307, -2.630769, -0.788313, 1.570796, 1.674520],accel_mss,speed_ms,0,blend_radius_m)
    movel([0.103804, -1.293583, -2.630608, -0.788198, 1.570796, 1.674600],accel_mss,speed_ms,0,blend_radius_m)
    movel([0.103792, -1.293977, -2.630377, -0.788035, 1.570796, 1.674589],accel_mss,speed_ms,0,blend_radius_m)
    movel([0.103523, -1.294338, -2.630165, -0.787886, 1.570796, 1.674319],accel_mss,speed_ms,0,blend_radius_m)
    movel([0.103297, -1.294618, -2.630001, -0.787771, 1.570796, 1.674094],accel_mss,speed_ms,0,blend_radius_m)
    movel([0.102982, -1.294687, -2.629960, -0.787742, 1.570796, 1.673778],accel_mss,speed_ms,0,blend_radius_m)
    movel([0.102668, -1.294988, -2.629783, -0.787618, 1.570796, 1.673465],accel_mss,speed_ms,0,blend_radius_m)
    movel([0.102281, -1.295194, -2.629662, -0.787533, 1.570796, 1.673077],accel_mss,speed_ms,0,blend_radius_m)
    movel([0.101902, -1.295350, -2.629570, -0.787469, 1.570796, 1.672698],accel_mss,speed_ms,0,blend_radius_m)
    movel([0.101557, -1.295489, -2.629488, -0.787412, 1.570796, 1.672353],accel_mss,speed_ms,0,blend_radius_m)
    movel([0.101243, -1.295617, -2.629413, -0.787359, 1.570796, 1.672039],accel_mss,speed_ms,0,blend_radius_m)
    movel([0.101286, -1.295842, -2.629280, -0.787267, 1.570796, 1.672083],accel_mss,speed_ms,0,blend_radius_m)
    movel([0.100997, -1.295991, -2.629193, -0.787206, 1.570796, 1.671793],accel_mss,speed_ms,0,blend_radius_m)
    movel([0.100718, -1.295951, -2.629216, -0.787222, 1.570796, 1.671514],accel_mss,speed_ms,0,blend_radius_m)
    movel([0.100425, -1.296077, -2.629142, -0.787170, 1.570796, 1.671222],accel_mss,speed_ms,0,blend_radius_m)
    movel([0.099331, -1.296580, -2.628845, -0.786964, 1.570796, 1.670127],accel_mss,speed_ms,0,blend_radius_m)
    movel([0.097242, -1.297292, -2.628425, -0.786672, 1.570796, 1.668038],accel_mss,speed_ms,0,blend_radius_m)
    movel([0.095038, -1.297963, -2.628028, -0.786398, 1.570796, 1.665834],accel_mss,speed_ms,0,blend_radius_m)
    movel([0.093267, -1.298398, -2.627770, -0.786220, 1.570796, 1.664064],accel_mss,speed_ms,0,blend_radius_m)
    movel([0.092796, -1.298507, -2.627706, -0.786176, 1.570796, 1.663592],accel_mss,speed_ms,0,blend_radius_m)
    movel([0.092505, -1.298577, -2.627664, -0.786148, 1.570796, 1.663301],accel_mss,speed_ms,0,blend_radius_m)
    movel([0.092006, -1.298695, -2.627594, -0.786099, 1.570796, 1.662802],accel_mss,speed_ms,0,blend_radius_m)
    movel([0.091686, -1.298709, -2.627586, -0.786094, 1.570796, 1.662483],accel_mss,speed_ms,0,blend_radius_m)
    movel([0.091516, -1.298549, -2.627681, -0.786159, 1.570796, 1.662312],accel_mss,speed_ms,0,blend_radius_m)
    movel([0.090908, -1.298604, -2.627648, -0.786137, 1.570796, 1.661704],accel_mss,speed_ms,0,blend_radius_m)
    movel([0.091012, -1.298791, -2.627537, -0.786060, 1.570796, 1.661808],accel_mss,speed_ms,0,blend_radius_m)
    movel([0.091131, -1.298957, -2.627439, -0.785993, 1.570796, 1.661927],accel_mss,speed_ms,0,blend_radius_m)
    movel([0.091380, -1.299030, -2.627396, -0.785963, 1.570796, 1.662176],accel_mss,speed_ms,0,blend_radius_m)
    movel([0.091703, -1.299034, -2.627394, -0.785962, 1.570796, 1.662500],accel_mss,speed_ms,0,blend_radius_m)
    movel([0.091970, -1.298785, -2.627541, -0.786063, 1.570796, 1.662766],accel_mss,speed_ms,0,blend_radius_m)
    movel([0.092331, -1.298807, -2.627528, -0.786054, 1.570796, 1.663127],accel_mss,speed_ms,0,blend_radius_m)
    movel([0.092659, -1.298717, -2.627581, -0.786090, 1.570796, 1.663455],accel_mss,speed_ms,0,blend_radius_m)
    movel([0.092762, -1.298900, -2.627473, -0.786016, 1.570796, 1.663559],accel_mss,speed_ms,0,blend_radius_m)
    movel([0.092991, -1.298961, -2.627436, -0.785991, 1.570796, 1.663787],accel_mss,speed_ms,0,blend_radius_m)
    movel([0.093296, -1.298783, -2.627542, -0.786064, 1.570796, 1.664092],accel_mss,speed_ms,0,blend_radius_m)
    movel([0.093554, -1.298769, -2.627551, -0.786070, 1.570796, 1.664350],accel_mss,speed_ms,0,blend_radius_m)
    movel([0.093259, -1.299029, -2.627397, -0.785964, 1.570796, 1.664056],accel_mss,speed_ms,0,blend_radius_m)
    movel([0.092956, -1.299112, -2.627347, -0.785930, 1.570796, 1.663753],accel_mss,speed_ms,0,blend_radius_m)
    movel([0.092691, -1.299070, -2.627372, -0.785947, 1.570796, 1.663487],accel_mss,speed_ms,0,blend_radius_m)
    movel([0.092356, -1.298978, -2.627427, -0.785984, 1.570796, 1.663152],accel_mss,speed_ms,0,blend_radius_m)
    movel([0.092063, -1.299023, -2.627400, -0.785966, 1.570796, 1.662859],accel_mss,speed_ms,0,blend_radius_m)
    movel([0.091652, -1.299143, -2.627329, -0.785917, 1.570796, 1.662448],accel_mss,speed_ms,0,blend_radius_m)
    movel([0.091327, -1.299231, -2.627276, -0.785881, 1.570796, 1.662123],accel_mss,speed_ms,0,blend_radius_m)
    movel([0.091035, -1.299288, -2.627243, -0.785858, 1.570796, 1.661832],accel_mss,speed_ms,0,blend_radius_m)
    movel([0.090721, -1.299331, -2.627217, -0.785841, 1.570796, 1.661517],accel_mss,speed_ms,0,blend_radius_m)
    movel([0.090684, -1.299094, -2.627358, -0.785937, 1.570796, 1.661480],accel_mss,speed_ms,0,blend_radius_m)
    movel([0.090510, -1.298965, -2.627434, -0.785990, 1.570796, 1.661306],accel_mss,speed_ms,0,blend_radius_m)
    movel([0.090188, -1.299079, -2.627367, -0.785943, 1.570796, 1.660984],accel_mss,speed_ms,0,blend_radius_m)
    movel([0.090012, -1.298940, -2.627449, -0.786000, 1.570796, 1.660808],accel_mss,speed_ms,0,blend_radius_m)
    movel([0.089943, -1.298729, -2.627574, -0.786086, 1.570796, 1.660739],accel_mss,speed_ms,0,blend_radius_m)
    movel([0.089712, -1.298679, -2.627604, -0.786106, 1.570796, 1.660509],accel_mss,speed_ms,0,blend_radius_m)
    movel([0.089970, -1.298437, -2.627747, -0.786205, 1.570796, 1.660766],accel_mss,speed_ms,0,blend_radius_m)
    movel([0.090285, -1.298394, -2.627773, -0.786222, 1.570796, 1.661081],accel_mss,speed_ms,0,blend_radius_m)
    movel([0.090132, -1.298683, -2.627602, -0.786105, 1.570796, 1.660928],accel_mss,speed_ms,0,blend_radius_m)
    movel([0.090205, -1.298963, -2.627436, -0.785991, 1.570796, 1.661001],accel_mss,speed_ms,0,blend_radius_m)
    movel([0.090261, -1.298678, -2.627605, -0.786107, 1.570796, 1.661057],accel_mss,speed_ms,0,blend_radius_m)
    movel([0.090563, -1.298554, -2.627678, -0.786157, 1.570796, 1.661359],accel_mss,speed_ms,0,blend_radius_m)
    movel([0.090470, -1.298342, -2.627804, -0.786244, 1.570796, 1.661266],accel_mss,speed_ms,0,blend_radius_m)
    movel([0.090383, -1.298068, -2.627966, -0.786355, 1.570796, 1.661179],accel_mss,speed_ms,0,blend_radius_m)
    movel([0.090678, -1.297826, -2.628109, -0.786454, 1.570796, 1.661474],accel_mss,speed_ms,0,blend_radius_m)
    movel([0.090825, -1.297494, -2.628306, -0.786590, 1.570796, 1.661621],accel_mss,speed_ms,0,blend_radius_m)
    movel([0.090518, -1.297690, -2.628189, -0.786509, 1.570796, 1.661314],accel_mss,speed_ms,0,blend_radius_m)
    movel([0.090290, -1.297927, -2.628049, -0.786413, 1.570796, 1.661086],accel_mss,speed_ms,0,blend_radius_m)
    movel([0.090113, -1.298212, -2.627880, -0.786296, 1.570796, 1.660910],accel_mss,speed_ms,0,blend_radius_m)
    movel([0.089804, -1.298280, -2.627840, -0.786269, 1.570796, 1.660600],accel_mss,speed_ms,0,blend_radius_m)
    movel([0.089954, -1.297963, -2.628028, -0.786398, 1.570796, 1.660750],accel_mss,speed_ms,0,blend_radius_m)
    movel([0.090167, -1.297691, -2.628189, -0.786509, 1.570796, 1.660963],accel_mss,speed_ms,0,blend_radius_m)
    movel([0.090457, -1.297347, -2.628392, -0.786650, 1.570796, 1.661253],accel_mss,speed_ms,0,blend_radius_m)
    movel([0.090350, -1.297056, -2.628564, -0.786769, 1.570796, 1.661146],accel_mss,speed_ms,0,blend_radius_m)
    movel([0.090002, -1.296971, -2.628614, -0.786803, 1.570796, 1.660798],accel_mss,speed_ms,0,blend_radius_m)
    movel([0.089628, -1.296935, -2.628635, -0.786818, 1.570796, 1.660424],accel_mss,speed_ms,0,blend_radius_m)
    movel([0.089304, -1.296977, -2.628611, -0.786801, 1.570796, 1.660101],accel_mss,speed_ms,0,blend_radius_m)
    movel([0.089032, -1.296934, -2.628637, -0.786819, 1.570796, 1.659829],accel_mss,speed_ms,0,blend_radius_m)
    movel([0.088749, -1.296974, -2.628613, -0.786802, 1.570796, 1.659546],accel_mss,speed_ms,0,blend_radius_m)
    movel([0.088519, -1.296916, -2.628647, -0.786826, 1.570796, 1.659315],accel_mss,speed_ms,0,blend_radius_m)
    movel([0.088260, -1.296793, -2.628720, -0.786877, 1.570796, 1.659057],accel_mss,speed_ms,0,blend_radius_m)
    movel([0.087984, -1.296604, -2.628831, -0.786954, 1.570796, 1.658780],accel_mss,speed_ms,0,blend_radius_m)
    movel([0.087838, -1.296402, -2.628950, -0.787037, 1.570796, 1.658634],accel_mss,speed_ms,0,blend_radius_m)
    movel([0.087930, -1.296130, -2.629111, -0.787148, 1.570796, 1.658726],accel_mss,speed_ms,0,blend_radius_m)
    movel([0.088018, -1.295835, -2.629284, -0.787270, 1.570796, 1.658814],accel_mss,speed_ms,0,blend_radius_m)
    movel([0.088177, -1.295298, -2.629600, -0.787490, 1.570796, 1.658973],accel_mss,speed_ms,0,blend_radius_m)
    movel([0.088520, -1.294882, -2.629845, -0.787662, 1.570796, 1.659316],accel_mss,speed_ms,0,blend_radius_m)
    movel([0.088850, -1.294590, -2.630017, -0.787782, 1.570796, 1.659647],accel_mss,speed_ms,0,blend_radius_m)
    movel([0.089096, -1.294365, -2.630149, -0.787875, 1.570796, 1.659893],accel_mss,speed_ms,0,blend_radius_m)
    movel([0.089150, -1.293993, -2.630367, -0.788029, 1.570796, 1.659946],accel_mss,speed_ms,0,blend_radius_m)
    movel([0.088850, -1.293957, -2.630389, -0.788044, 1.570796, 1.659646],accel_mss,speed_ms,0,blend_radius_m)
    movel([0.088651, -1.293819, -2.630469, -0.788100, 1.570796, 1.659447],accel_mss,speed_ms,0,blend_radius_m)
    movel([0.088309, -1.293899, -2.630422, -0.788068, 1.570796, 1.659105],accel_mss,speed_ms,0,blend_radius_m)
    movel([0.087687, -1.293983, -2.630373, -0.788033, 1.570796, 1.658483],accel_mss,speed_ms,0,blend_radius_m)
    movel([0.087026, -1.293852, -2.630450, -0.788087, 1.570796, 1.657823],accel_mss,speed_ms,0,blend_radius_m)
    movel([0.086481, -1.293564, -2.630619, -0.788206, 1.570796, 1.657277],accel_mss,speed_ms,0,blend_radius_m)
    movel([0.086205, -1.293166, -2.630852, -0.788371, 1.570796, 1.657001],accel_mss,speed_ms,0,blend_radius_m)
    movel([0.086167, -1.292865, -2.631028, -0.788496, 1.570796, 1.656963],accel_mss,speed_ms,0,blend_radius_m)
    movel([0.086235, -1.292549, -2.631213, -0.788627, 1.570796, 1.657032],accel_mss,speed_ms,0,blend_radius_m)
    movel([0.086426, -1.292178, -2.631430, -0.788781, 1.570796, 1.657222],accel_mss,speed_ms,0,blend_radius_m)
    movel([0.086757, -1.291717, -2.631699, -0.788973, 1.570796, 1.657553],accel_mss,speed_ms,0,blend_radius_m)
    movel([0.086981, -1.291477, -2.631839, -0.789073, 1.570796, 1.657777],accel_mss,speed_ms,0,blend_radius_m)
    movel([0.087305, -1.291207, -2.631997, -0.789185, 1.570796, 1.658101],accel_mss,speed_ms,0,blend_radius_m)
    movel([0.087627, -1.290981, -2.632129, -0.789279, 1.570796, 1.658423],accel_mss,speed_ms,0,blend_radius_m)
    movel([0.087930, -1.290792, -2.632238, -0.789358, 1.570796, 1.658726],accel_mss,speed_ms,0,blend_radius_m)
    movel([0.088216, -1.290788, -2.632241, -0.789360, 1.570796, 1.659013],accel_mss,speed_ms,0,blend_radius_m)
    movel([0.088406, -1.290922, -2.632163, -0.789304, 1.570796, 1.659202],accel_mss,speed_ms,0,blend_radius_m)
    movel([0.088248, -1.290579, -2.632363, -0.789447, 1.570796, 1.659044],accel_mss,speed_ms,0,blend_radius_m)
    movel([0.088513, -1.290389, -2.632473, -0.789526, 1.570796, 1.659309],accel_mss,speed_ms,0,blend_radius_m)
    movel([0.088853, -1.290071, -2.632658, -0.789660, 1.570796, 1.659650],accel_mss,speed_ms,0,blend_radius_m)
    movel([0.089467, -1.289643, -2.632907, -0.789839, 1.570796, 1.660263],accel_mss,speed_ms,0,blend_radius_m)
    movel([0.090092, -1.289248, -2.633137, -0.790004, 1.570796, 1.660888],accel_mss,speed_ms,0,blend_radius_m)
    movel([0.090426, -1.289175, -2.633179, -0.790035, 1.570796, 1.661223],accel_mss,speed_ms,0,blend_radius_m)
    movel([0.090517, -1.289419, -2.633037, -0.789932, 1.570796, 1.661314],accel_mss,speed_ms,0,blend_radius_m)
    speed_ms = 0.003
    movel([0.090517, -1.275491, -2.626410, -0.810488, 1.570796, 1.661314],accel_mss,speed_ms,0,blend_radius_m)
    speed_ms = 1.000
    movel([0.090517, -1.248993, -2.612771, -0.850625, 1.570796, 1.661314],accel_mss,speed_ms,0,blend_radius_m)
    movel([0.108394, -1.243984, -2.615506, -0.852900, 1.570796, 1.679191],accel_mss,speed_ms,0,blend_radius_m)
    movel([0.108394, -1.270545, -2.629211, -0.812633, 1.570796, 1.679191],accel_mss,speed_ms,0,blend_radius_m)
    speed_ms = 0.003
    movel([0.108394, -1.280978, -2.634218, -0.797193, 1.570796, 1.679191],accel_mss,speed_ms,0,blend_radius_m)
    speed_ms = 0.007
    movel([0.108672, -1.280919, -2.634252, -0.797218, 1.570796, 1.679468],accel_mss,speed_ms,0,blend_radius_m)
    movel([0.108972, -1.280870, -2.634280, -0.797239, 1.570796, 1.679768],accel_mss,speed_ms,0,blend_radius_m)
    movel([0.108590, -1.281076, -2.634162, -0.797151, 1.570796, 1.679387],accel_mss,speed_ms,0,blend_radius_m)
    movel([0.108394, -1.280978, -2.634218, -0.797193, 1.570796, 1.679191],accel_mss,speed_ms,0,blend_radius_m)
    speed_ms = 0.003
    movel([0.108394, -1.284514, -2.635871, -0.792004, 1.570796, 1.679191],accel_mss,speed_ms,0,blend_radius_m)
    speed_ms = 0.007
    movel([0.108672, -1.284455, -2.635905, -0.792029, 1.570796, 1.679468],accel_mss,speed_ms,0,blend_radius_m)
    movel([0.108972, -1.284406, -2.635933, -0.792050, 1.570796, 1.679768],accel_mss,speed_ms,0,blend_radius_m)
    movel([0.108590, -1.284612, -2.635815, -0.791962, 1.570796, 1.679387],accel_mss,speed_ms,0,blend_radius_m)
    movel([0.108394, -1.284514, -2.635871, -0.792004, 1.570796, 1.679191],accel_mss,speed_ms,0,blend_radius_m)
    speed_ms = 0.003
    movel([0.108394, -1.270545, -2.629211, -0.812633, 1.570796, 1.679191],accel_mss,speed_ms,0,blend_radius_m)
    speed_ms = 1.000
    movel([0.108394, -1.243984, -2.615506, -0.852900, 1.570796, 1.679191],accel_mss,speed_ms,0,blend_radius_m)
    movel([0.134199, -1.228063, -2.624004, -0.860322, 1.570796, 1.704996],accel_mss,speed_ms,0,blend_radius_m)
    movel([0.134199, -1.254817, -2.637919, -0.819653, 1.570796, 1.704996],accel_mss,speed_ms,0,blend_radius_m)
    speed_ms = 0.003
    movel([0.134199, -1.265339, -2.643007, -0.804044, 1.570796, 1.704996],accel_mss,speed_ms,0,blend_radius_m)
    speed_ms = 0.007
    movel([0.134398, -1.265029, -2.643178, -0.804183, 1.570796, 1.705194],accel_mss,speed_ms,0,blend_radius_m)
    movel([0.134745, -1.264784, -2.643313, -0.804292, 1.570796, 1.705541],accel_mss,speed_ms,0,blend_radius_m)
    movel([0.135237, -1.264642, -2.643391, -0.804356, 1.570796, 1.706033],accel_mss,speed_ms,0,blend_radius_m)
    movel([0.135651, -1.264639, -2.643393, -0.804357, 1.570796, 1.706448],accel_mss,speed_ms,0,blend_radius_m)
    movel([0.135748, -1.264848, -2.643278, -0.804264, 1.570796, 1.706545],accel_mss,speed_ms,0,blend_radius_m)
    movel([0.135483, -1.265183, -2.643092, -0.804113, 1.570796, 1.706279],accel_mss,speed_ms,0,blend_radius_m)
    movel([0.135213, -1.265424, -2.642960, -0.804005, 1.570796, 1.706009],accel_mss,speed_ms,0,blend_radius_m)
    movel([0.134898, -1.265584, -2.642871, -0.803934, 1.570796, 1.705694],accel_mss,speed_ms,0,blend_radius_m)
    movel([0.134599, -1.265633, -2.642844, -0.803912, 1.570796, 1.705396],accel_mss,speed_ms,0,blend_radius_m)
    movel([0.134371, -1.265561, -2.642884, -0.803944, 1.570796, 1.705167],accel_mss,speed_ms,0,blend_radius_m)
    movel([0.134199, -1.265339, -2.643007, -0.804044, 1.570796, 1.704996],accel_mss,speed_ms,0,blend_radius_m)
    speed_ms = 0.003
    movel([0.134199, -1.268907, -2.644686, -0.798796, 1.570796, 1.704996],accel_mss,speed_ms,0,blend_radius_m)
    speed_ms = 0.007
    movel([0.134398, -1.268597, -2.644858, -0.798934, 1.570796, 1.705194],accel_mss,speed_ms,0,blend_radius_m)
    movel([0.134745, -1.268352, -2.644993, -0.799043, 1.570796, 1.705541],accel_mss,speed_ms,0,blend_radius_m)
    movel([0.135237, -1.268211, -2.645072, -0.799106, 1.570796, 1.706033],accel_mss,speed_ms,0,blend_radius_m)
    movel([0.135651, -1.268209, -2.645073, -0.799107, 1.570796, 1.706448],accel_mss,speed_ms,0,blend_radius_m)
    movel([0.135748, -1.268416, -2.644958, -0.799015, 1.570796, 1.706545],accel_mss,speed_ms,0,blend_radius_m)
    movel([0.135483, -1.268752, -2.644772, -0.798865, 1.570796, 1.706279],accel_mss,speed_ms,0,blend_radius_m)
    movel([0.135213, -1.268992, -2.644639, -0.798758, 1.570796, 1.706009],accel_mss,speed_ms,0,blend_radius_m)
    movel([0.134898, -1.269152, -2.644550, -0.798687, 1.570796, 1.705694],accel_mss,speed_ms,0,blend_radius_m)
    movel([0.134599, -1.269200, -2.644523, -0.798666, 1.570796, 1.705396],accel_mss,speed_ms,0,blend_radius_m)
    movel([0.134371, -1.269128, -2.644563, -0.798698, 1.570796, 1.705167],accel_mss,speed_ms,0,blend_radius_m)
    movel([0.134199, -1.268907, -2.644686, -0.798796, 1.570796, 1.704996],accel_mss,speed_ms,0,blend_radius_m)
    speed_ms = 0.003
    movel([0.134199, -1.254817, -2.637919, -0.819653, 1.570796, 1.704996],accel_mss,speed_ms,0,blend_radius_m)
    speed_ms = 1.000
    movel([0.134199, -1.228063, -2.624004, -0.860322, 1.570796, 1.704996],accel_mss,speed_ms,0,blend_radius_m)
    movel([0.135018, -1.226764, -2.624685, -0.860940, 1.570796, 1.705815],accel_mss,speed_ms,0,blend_radius_m)
    movel([0.135018, -1.253533, -2.638617, -0.820240, 1.570796, 1.705815],accel_mss,speed_ms,0,blend_radius_m)
    speed_ms = 0.003
    movel([0.135018, -1.264062, -2.643711, -0.804616, 1.570796, 1.705815],accel_mss,speed_ms,0,blend_radius_m)
    speed_ms = 0.007
    movel([0.133569, -1.264514, -2.643462, -0.804413, 1.570796, 1.704366],accel_mss,speed_ms,0,blend_radius_m)
    movel([0.132754, -1.264606, -2.643411, -0.804372, 1.570796, 1.703551],accel_mss,speed_ms,0,blend_radius_m)
    movel([0.132393, -1.264541, -2.643447, -0.804401, 1.570796, 1.703189],accel_mss,speed_ms,0,blend_radius_m)
    movel([0.132220, -1.264399, -2.643525, -0.804465, 1.570796, 1.703016],accel_mss,speed_ms,0,blend_radius_m)
    movel([0.132406, -1.263908, -2.643795, -0.804685, 1.570796, 1.703203],accel_mss,speed_ms,0,blend_radius_m)
    movel([0.132616, -1.263631, -2.643948, -0.804810, 1.570796, 1.703412],accel_mss,speed_ms,0,blend_radius_m)
    movel([0.132602, -1.263320, -2.644119, -0.804950, 1.570796, 1.703398],accel_mss,speed_ms,0,blend_radius_m)
    movel([0.132363, -1.263216, -2.644176, -0.804997, 1.570796, 1.703159],accel_mss,speed_ms,0,blend_radius_m)
    movel([0.132010, -1.263108, -2.644235, -0.805045, 1.570796, 1.702806],accel_mss,speed_ms,0,blend_radius_m)
    movel([0.132437, -1.262707, -2.644456, -0.805226, 1.570796, 1.703234],accel_mss,speed_ms,0,blend_radius_m)
    movel([0.132758, -1.262384, -2.644633, -0.805372, 1.570796, 1.703554],accel_mss,speed_ms,0,blend_radius_m)
    movel([0.132813, -1.262065, -2.644808, -0.805516, 1.570796, 1.703609],accel_mss,speed_ms,0,blend_radius_m)
    movel([0.132580, -1.261897, -2.644900, -0.805592, 1.570796, 1.703377],accel_mss,speed_ms,0,blend_radius_m)
    movel([0.132378, -1.261707, -2.645004, -0.805678, 1.570796, 1.703175],accel_mss,speed_ms,0,blend_radius_m)
    movel([0.132314, -1.261470, -2.645134, -0.805785, 1.570796, 1.703111],accel_mss,speed_ms,0,blend_radius_m)
    movel([0.132399, -1.261194, -2.645285, -0.805910, 1.570796, 1.703195],accel_mss,speed_ms,0,blend_radius_m)
    movel([0.132615, -1.260893, -2.645450, -0.806046, 1.570796, 1.703411],accel_mss,speed_ms,0,blend_radius_m)
    movel([0.132980, -1.260625, -2.645596, -0.806168, 1.570796, 1.703776],accel_mss,speed_ms,0,blend_radius_m)
    movel([0.133606, -1.260445, -2.645695, -0.806250, 1.570796, 1.704403],accel_mss,speed_ms,0,blend_radius_m)
    movel([0.134003, -1.260357, -2.645743, -0.806289, 1.570796, 1.704799],accel_mss,speed_ms,0,blend_radius_m)
    movel([0.134688, -1.260200, -2.645828, -0.806361, 1.570796, 1.705485],accel_mss,speed_ms,0,blend_radius_m)
    movel([0.135480, -1.260013, -2.645930, -0.806446, 1.570796, 1.706276],accel_mss,speed_ms,0,blend_radius_m)
    movel([0.136283, -1.259823, -2.646034, -0.806532, 1.570796, 1.707080],accel_mss,speed_ms,0,blend_radius_m)
    movel([0.137293, -1.259591, -2.646161, -0.806637, 1.570796, 1.708089],accel_mss,speed_ms,0,blend_radius_m)
    movel([0.137906, -1.259479, -2.646222, -0.806688, 1.570796, 1.708703],accel_mss,speed_ms,0,blend_radius_m)
    movel([0.138308, -1.259446, -2.646240, -0.806703, 1.570796, 1.709104],accel_mss,speed_ms,0,blend_radius_m)
    movel([0.138558, -1.259495, -2.646213, -0.806681, 1.570796, 1.709354],accel_mss,speed_ms,0,blend_radius_m)
    movel([0.138772, -1.259631, -2.646139, -0.806619, 1.570796, 1.709569],accel_mss,speed_ms,0,blend_radius_m)
    movel([0.138742, -1.260008, -2.645933, -0.806448, 1.570796, 1.709538],accel_mss,speed_ms,0,blend_radius_m)
    movel([0.138459, -1.260449, -2.645692, -0.806248, 1.570796, 1.709255],accel_mss,speed_ms,0,blend_radius_m)
    movel([0.138261, -1.260761, -2.645522, -0.806106, 1.570796, 1.709057],accel_mss,speed_ms,0,blend_radius_m)
    movel([0.138159, -1.261142, -2.645313, -0.805933, 1.570796, 1.708956],accel_mss,speed_ms,0,blend_radius_m)
    movel([0.138212, -1.261391, -2.645178, -0.805821, 1.570796, 1.709008],accel_mss,speed_ms,0,blend_radius_m)
    movel([0.138231, -1.261781, -2.644964, -0.805644, 1.570796, 1.709028],accel_mss,speed_ms,0,blend_radius_m)
    movel([0.138086, -1.262178, -2.644746, -0.805465, 1.570796, 1.708883],accel_mss,speed_ms,0,blend_radius_m)
    movel([0.137764, -1.262595, -2.644517, -0.805277, 1.570796, 1.708560],accel_mss,speed_ms,0,blend_radius_m)
    movel([0.137253, -1.263048, -2.644269, -0.805072, 1.570796, 1.708050],accel_mss,speed_ms,0,blend_radius_m)
    movel([0.136472, -1.263511, -2.644014, -0.804864, 1.570796, 1.707268],accel_mss,speed_ms,0,blend_radius_m)
    movel([0.135018, -1.264062, -2.643711, -0.804616, 1.570796, 1.705815],accel_mss,speed_ms,0,blend_radius_m)
    speed_ms = 0.003
    movel([0.135018, -1.267632, -2.645392, -0.799364, 1.570796, 1.705815],accel_mss,speed_ms,0,blend_radius_m)
    speed_ms = 0.007
    movel([0.133569, -1.268083, -2.645143, -0.799163, 1.570796, 1.704366],accel_mss,speed_ms,0,blend_radius_m)
    movel([0.132754, -1.268175, -2.645092, -0.799122, 1.570796, 1.703551],accel_mss,speed_ms,0,blend_radius_m)
    movel([0.132393, -1.268110, -2.645128, -0.799151, 1.570796, 1.703189],accel_mss,speed_ms,0,blend_radius_m)
    movel([0.132220, -1.267969, -2.645206, -0.799214, 1.570796, 1.703016],accel_mss,speed_ms,0,blend_radius_m)
    movel([0.132406, -1.267479, -2.645477, -0.799433, 1.570796, 1.703203],accel_mss,speed_ms,0,blend_radius_m)
    movel([0.132616, -1.267202, -2.645630, -0.799557, 1.570796, 1.703412],accel_mss,speed_ms,0,blend_radius_m)
    movel([0.132602, -1.266891, -2.645802, -0.799695, 1.570796, 1.703398],accel_mss,speed_ms,0,blend_radius_m)
    movel([0.132363, -1.266788, -2.645859, -0.799742, 1.570796, 1.703159],accel_mss,speed_ms,0,blend_radius_m)
    movel([0.132010, -1.266681, -2.645919, -0.799790, 1.570796, 1.702806],accel_mss,speed_ms,0,blend_radius_m)
    movel([0.132437, -1.266280, -2.646140, -0.799969, 1.570796, 1.703234],accel_mss,speed_ms,0,blend_radius_m)
    movel([0.132758, -1.265958, -2.646318, -0.800114, 1.570796, 1.703554],accel_mss,speed_ms,0,blend_radius_m)
    movel([0.132813, -1.265640, -2.646493, -0.800256, 1.570796, 1.703609],accel_mss,speed_ms,0,blend_radius_m)
    movel([0.132580, -1.265472, -2.646585, -0.800332, 1.570796, 1.703377],accel_mss,speed_ms,0,blend_radius_m)
    movel([0.132378, -1.265282, -2.646690, -0.800417, 1.570796, 1.703175],accel_mss,speed_ms,0,blend_radius_m)
    movel([0.132314, -1.265045, -2.646820, -0.800523, 1.570796, 1.703111],accel_mss,speed_ms,0,blend_radius_m)
    movel([0.132399, -1.264770, -2.646972, -0.800647, 1.570796, 1.703195],accel_mss,speed_ms,0,blend_radius_m)
    movel([0.132615, -1.264470, -2.647137, -0.800782, 1.570796, 1.703411],accel_mss,speed_ms,0,blend_radius_m)
    movel([0.132980, -1.264202, -2.647284, -0.800903, 1.570796, 1.703776],accel_mss,speed_ms,0,blend_radius_m)
    movel([0.133606, -1.264022, -2.647383, -0.800984, 1.570796, 1.704403],accel_mss,speed_ms,0,blend_radius_m)
    movel([0.134003, -1.263934, -2.647431, -0.801024, 1.570796, 1.704799],accel_mss,speed_ms,0,blend_radius_m)
    movel([0.134688, -1.263778, -2.647517, -0.801094, 1.570796, 1.705485],accel_mss,speed_ms,0,blend_radius_m)
    movel([0.135480, -1.263591, -2.647619, -0.801179, 1.570796, 1.706276],accel_mss,speed_ms,0,blend_radius_m)
    movel([0.136283, -1.263401, -2.647723, -0.801264, 1.570796, 1.707080],accel_mss,speed_ms,0,blend_radius_m)
    movel([0.137293, -1.263170, -2.647850, -0.801369, 1.570796, 1.708089],accel_mss,speed_ms,0,blend_radius_m)
    movel([0.137906, -1.263058, -2.647911, -0.801420, 1.570796, 1.708703],accel_mss,speed_ms,0,blend_radius_m)
    movel([0.138308, -1.263025, -2.647930, -0.801435, 1.570796, 1.709104],accel_mss,speed_ms,0,blend_radius_m)
    movel([0.138558, -1.263074, -2.647902, -0.801412, 1.570796, 1.709354],accel_mss,speed_ms,0,blend_radius_m)
    movel([0.138772, -1.263210, -2.647828, -0.801351, 1.570796, 1.709569],accel_mss,speed_ms,0,blend_radius_m)
    movel([0.138742, -1.263586, -2.647622, -0.801181, 1.570796, 1.709538],accel_mss,speed_ms,0,blend_radius_m)
    movel([0.138459, -1.264027, -2.647380, -0.800982, 1.570796, 1.709255],accel_mss,speed_ms,0,blend_radius_m)
    movel([0.138261, -1.264338, -2.647209, -0.800842, 1.570796, 1.709057],accel_mss,speed_ms,0,blend_radius_m)
    movel([0.138159, -1.264718, -2.647000, -0.800671, 1.570796, 1.708956],accel_mss,speed_ms,0,blend_radius_m)
    movel([0.138212, -1.264966, -2.646864, -0.800559, 1.570796, 1.709008],accel_mss,speed_ms,0,blend_radius_m)
    movel([0.138231, -1.265356, -2.646649, -0.800384, 1.570796, 1.709028],accel_mss,speed_ms,0,blend_radius_m)
    movel([0.138086, -1.265752, -2.646431, -0.800206, 1.570796, 1.708883],accel_mss,speed_ms,0,blend_radius_m)
    movel([0.137764, -1.266168, -2.646201, -0.800019, 1.570796, 1.708560],accel_mss,speed_ms,0,blend_radius_m)
    movel([0.137253, -1.266620, -2.645952, -0.799817, 1.570796, 1.708050],accel_mss,speed_ms,0,blend_radius_m)
    movel([0.136472, -1.267082, -2.645697, -0.799610, 1.570796, 1.707268],accel_mss,speed_ms,0,blend_radius_m)
    movel([0.135018, -1.267632, -2.645392, -0.799364, 1.570796, 1.705815],accel_mss,speed_ms,0,blend_radius_m)
    speed_ms = 0.003
    movel([0.135018, -1.253533, -2.638617, -0.820240, 1.570796, 1.705815],accel_mss,speed_ms,0,blend_radius_m)
    speed_ms = 1.000
    movel([0.135018, -1.226764, -2.624685, -0.860940, 1.570796, 1.705815],accel_mss,speed_ms,0,blend_radius_m)
    movel([0.137358, -1.221519, -2.627413, -0.863457, 1.570796, 1.708154],accel_mss,speed_ms,0,blend_radius_m)
    movel([0.137358, -1.248347, -2.641414, -0.822628, 1.570796, 1.708154],accel_mss,speed_ms,0,blend_radius_m)
    speed_ms = 0.003
    movel([0.137358, -1.258904, -2.646535, -0.806950, 1.570796, 1.708154],accel_mss,speed_ms,0,blend_radius_m)
    speed_ms = 0.007
    movel([0.137144, -1.258616, -2.646692, -0.807081, 1.570796, 1.707940],accel_mss,speed_ms,0,blend_radius_m)
    movel([0.137235, -1.257961, -2.647048, -0.807380, 1.570796, 1.708031],accel_mss,speed_ms,0,blend_radius_m)
    movel([0.137436, -1.256880, -2.647634, -0.807874, 1.570796, 1.708233],accel_mss,speed_ms,0,blend_radius_m)
    movel([0.137871, -1.254806, -2.648756, -0.808827, 1.570796, 1.708667],accel_mss,speed_ms,0,blend_radius_m)
    movel([0.138200, -1.253306, -2.649563, -0.809519, 1.570796, 1.708997],accel_mss,speed_ms,0,blend_radius_m)
    movel([0.138501, -1.252015, -2.650256, -0.810117, 1.570796, 1.709297],accel_mss,speed_ms,0,blend_radius_m)
    movel([0.138778, -1.250887, -2.650861, -0.810642, 1.570796, 1.709574],accel_mss,speed_ms,0,blend_radius_m)
    movel([0.139175, -1.250471, -2.651083, -0.810835, 1.570796, 1.709971],accel_mss,speed_ms,0,blend_radius_m)
    movel([0.139446, -1.250254, -2.651199, -0.810936, 1.570796, 1.710242],accel_mss,speed_ms,0,blend_radius_m)
    movel([0.139737, -1.250029, -2.651319, -0.811041, 1.570796, 1.710534],accel_mss,speed_ms,0,blend_radius_m)
    movel([0.140340, -1.249523, -2.651589, -0.811277, 1.570796, 1.711136],accel_mss,speed_ms,0,blend_radius_m)
    movel([0.140778, -1.249049, -2.651841, -0.811499, 1.570796, 1.711574],accel_mss,speed_ms,0,blend_radius_m)
    movel([0.141088, -1.248562, -2.652101, -0.811727, 1.570796, 1.711885],accel_mss,speed_ms,0,blend_radius_m)
    movel([0.141299, -1.248024, -2.652387, -0.811978, 1.570796, 1.712095],accel_mss,speed_ms,0,blend_radius_m)
    movel([0.141376, -1.247686, -2.652566, -0.812137, 1.570796, 1.712172],accel_mss,speed_ms,0,blend_radius_m)
    movel([0.141270, -1.247330, -2.652755, -0.812304, 1.570796, 1.712067],accel_mss,speed_ms,0,blend_radius_m)
    movel([0.141024, -1.247133, -2.652860, -0.812396, 1.570796, 1.711820],accel_mss,speed_ms,0,blend_radius_m)
    movel([0.140322, -1.246938, -2.652963, -0.812488, 1.570796, 1.711118],accel_mss,speed_ms,0,blend_radius_m)
    movel([0.139577, -1.247221, -2.652813, -0.812355, 1.570796, 1.710374],accel_mss,speed_ms,0,blend_radius_m)
    movel([0.138926, -1.247946, -2.652428, -0.812015, 1.570796, 1.709723],accel_mss,speed_ms,0,blend_radius_m)
    movel([0.138497, -1.248983, -2.651876, -0.811529, 1.570796, 1.709294],accel_mss,speed_ms,0,blend_radius_m)
    movel([0.138299, -1.249669, -2.651511, -0.811209, 1.570796, 1.709096],accel_mss,speed_ms,0,blend_radius_m)
    movel([0.138115, -1.250027, -2.651320, -0.811042, 1.570796, 1.708911],accel_mss,speed_ms,0,blend_radius_m)
    movel([0.137451, -1.250470, -2.651084, -0.810836, 1.570796, 1.708247],accel_mss,speed_ms,0,blend_radius_m)
    movel([0.137003, -1.250600, -2.651014, -0.810775, 1.570796, 1.707799],accel_mss,speed_ms,0,blend_radius_m)
    movel([0.136737, -1.250566, -2.651032, -0.810791, 1.570796, 1.707533],accel_mss,speed_ms,0,blend_radius_m)
    movel([0.136577, -1.250358, -2.651143, -0.810888, 1.570796, 1.707374],accel_mss,speed_ms,0,blend_radius_m)
    movel([0.136485, -1.249888, -2.651394, -0.811107, 1.570796, 1.707281],accel_mss,speed_ms,0,blend_radius_m)
    movel([0.136093, -1.248988, -2.651874, -0.811527, 1.570796, 1.706889],accel_mss,speed_ms,0,blend_radius_m)
    movel([0.135259, -1.248595, -2.652083, -0.811711, 1.570796, 1.706056],accel_mss,speed_ms,0,blend_radius_m)
    movel([0.134232, -1.248815, -2.651966, -0.811608, 1.570796, 1.705028],accel_mss,speed_ms,0,blend_radius_m)
    movel([0.133293, -1.249559, -2.651569, -0.811260, 1.570796, 1.704090],accel_mss,speed_ms,0,blend_radius_m)
    movel([0.132861, -1.250341, -2.651152, -0.810896, 1.570796, 1.703657],accel_mss,speed_ms,0,blend_radius_m)
    movel([0.132871, -1.251012, -2.650794, -0.810583, 1.570796, 1.703667],accel_mss,speed_ms,0,blend_radius_m)
    movel([0.133354, -1.251468, -2.650550, -0.810371, 1.570796, 1.704151],accel_mss,speed_ms,0,blend_radius_m)
    movel([0.134238, -1.251642, -2.650456, -0.810290, 1.570796, 1.705035],accel_mss,speed_ms,0,blend_radius_m)
    movel([0.134548, -1.251641, -2.650457, -0.810291, 1.570796, 1.705344],accel_mss,speed_ms,0,blend_radius_m)
    movel([0.134854, -1.251627, -2.650465, -0.810298, 1.570796, 1.705650],accel_mss,speed_ms,0,blend_radius_m)
    movel([0.135274, -1.251568, -2.650496, -0.810325, 1.570796, 1.706071],accel_mss,speed_ms,0,blend_radius_m)
    movel([0.135532, -1.251584, -2.650487, -0.810317, 1.570796, 1.706328],accel_mss,speed_ms,0,blend_radius_m)
    movel([0.135756, -1.251751, -2.650398, -0.810240, 1.570796, 1.706552],accel_mss,speed_ms,0,blend_radius_m)
    movel([0.135846, -1.252036, -2.650246, -0.810108, 1.570796, 1.706642],accel_mss,speed_ms,0,blend_radius_m)
    movel([0.135832, -1.252571, -2.649958, -0.809860, 1.570796, 1.706628],accel_mss,speed_ms,0,blend_radius_m)
    movel([0.135724, -1.253517, -2.649450, -0.809422, 1.570796, 1.706520],accel_mss,speed_ms,0,blend_radius_m)
    movel([0.135420, -1.255572, -2.648342, -0.808475, 1.570796, 1.706217],accel_mss,speed_ms,0,blend_radius_m)
    movel([0.135034, -1.258058, -2.646995, -0.807336, 1.570796, 1.705830],accel_mss,speed_ms,0,blend_radius_m)
    movel([0.134814, -1.258982, -2.646492, -0.806914, 1.570796, 1.705611],accel_mss,speed_ms,0,blend_radius_m)
    movel([0.134542, -1.259451, -2.646237, -0.806701, 1.570796, 1.705338],accel_mss,speed_ms,0,blend_radius_m)
    movel([0.134131, -1.259731, -2.646084, -0.806574, 1.570796, 1.704927],accel_mss,speed_ms,0,blend_radius_m)
    movel([0.133824, -1.259748, -2.646075, -0.806566, 1.570796, 1.704620],accel_mss,speed_ms,0,blend_radius_m)
    movel([0.133658, -1.259591, -2.646161, -0.806637, 1.570796, 1.704454],accel_mss,speed_ms,0,blend_radius_m)
    movel([0.133614, -1.259182, -2.646384, -0.806824, 1.570796, 1.704411],accel_mss,speed_ms,0,blend_radius_m)
    movel([0.133693, -1.258313, -2.646857, -0.807220, 1.570796, 1.704489],accel_mss,speed_ms,0,blend_radius_m)
    movel([0.133760, -1.257672, -2.647205, -0.807512, 1.570796, 1.704556],accel_mss,speed_ms,0,blend_radius_m)
    movel([0.133768, -1.257296, -2.647409, -0.807684, 1.570796, 1.704565],accel_mss,speed_ms,0,blend_radius_m)
    movel([0.133641, -1.257005, -2.647567, -0.807817, 1.570796, 1.704437],accel_mss,speed_ms,0,blend_radius_m)
    movel([0.133135, -1.257023, -2.647557, -0.807809, 1.570796, 1.703932],accel_mss,speed_ms,0,blend_radius_m)
    movel([0.132693, -1.257059, -2.647538, -0.807793, 1.570796, 1.703489],accel_mss,speed_ms,0,blend_radius_m)
    movel([0.132205, -1.257107, -2.647512, -0.807771, 1.570796, 1.703001],accel_mss,speed_ms,0,blend_radius_m)
    movel([0.131165, -1.257148, -2.647489, -0.807752, 1.570796, 1.701961],accel_mss,speed_ms,0,blend_radius_m)
    movel([0.130280, -1.257046, -2.647545, -0.807799, 1.570796, 1.701076],accel_mss,speed_ms,0,blend_radius_m)
    movel([0.129498, -1.256778, -2.647690, -0.807922, 1.570796, 1.700295],accel_mss,speed_ms,0,blend_radius_m)
    movel([0.128756, -1.256342, -2.647926, -0.808121, 1.570796, 1.699553],accel_mss,speed_ms,0,blend_radius_m)
    movel([0.127629, -1.254975, -2.648665, -0.808749, 1.570796, 1.698425],accel_mss,speed_ms,0,blend_radius_m)
    movel([0.127239, -1.253124, -2.649661, -0.809604, 1.570796, 1.698036],accel_mss,speed_ms,0,blend_radius_m)
    movel([0.127630, -1.250874, -2.650868, -0.810648, 1.570796, 1.698426],accel_mss,speed_ms,0,blend_radius_m)
    movel([0.128781, -1.248347, -2.652215, -0.811827, 1.570796, 1.699577],accel_mss,speed_ms,0,blend_radius_m)
    movel([0.129174, -1.247712, -2.652552, -0.812125, 1.570796, 1.699970],accel_mss,speed_ms,0,blend_radius_m)
    movel([0.129602, -1.247109, -2.652872, -0.812408, 1.570796, 1.700398],accel_mss,speed_ms,0,blend_radius_m)
    movel([0.130119, -1.246465, -2.653213, -0.812710, 1.570796, 1.700916],accel_mss,speed_ms,0,blend_radius_m)
    movel([0.130785, -1.245709, -2.653613, -0.813066, 1.570796, 1.701581],accel_mss,speed_ms,0,blend_radius_m)
    movel([0.132478, -1.244039, -2.654494, -0.813856, 1.570796, 1.703274],accel_mss,speed_ms,0,blend_radius_m)
    movel([0.134231, -1.242693, -2.655202, -0.814494, 1.570796, 1.705028],accel_mss,speed_ms,0,blend_radius_m)
    movel([0.136117, -1.241632, -2.655759, -0.814999, 1.570796, 1.706913],accel_mss,speed_ms,0,blend_radius_m)
    movel([0.138201, -1.240803, -2.656192, -0.815394, 1.570796, 1.708998],accel_mss,speed_ms,0,blend_radius_m)
    movel([0.139435, -1.240437, -2.656383, -0.815568, 1.570796, 1.710232],accel_mss,speed_ms,0,blend_radius_m)
    movel([0.140458, -1.240212, -2.656501, -0.815676, 1.570796, 1.711255],accel_mss,speed_ms,0,blend_radius_m)
    movel([0.141377, -1.240102, -2.656558, -0.815729, 1.570796, 1.712174],accel_mss,speed_ms,0,blend_radius_m)
    movel([0.142291, -1.240094, -2.656562, -0.815732, 1.570796, 1.713088],accel_mss,speed_ms,0,blend_radius_m)
    movel([0.144324, -1.240459, -2.656372, -0.815558, 1.570796, 1.715120],accel_mss,speed_ms,0,blend_radius_m)
    movel([0.145972, -1.241324, -2.655920, -0.815145, 1.570796, 1.716769],accel_mss,speed_ms,0,blend_radius_m)
    movel([0.147123, -1.242616, -2.655243, -0.814531, 1.570796, 1.717920],accel_mss,speed_ms,0,blend_radius_m)
    movel([0.147683, -1.244233, -2.654392, -0.813764, 1.570796, 1.718479],accel_mss,speed_ms,0,blend_radius_m)
    movel([0.147706, -1.244999, -2.653988, -0.813402, 1.570796, 1.718502],accel_mss,speed_ms,0,blend_radius_m)
    movel([0.147581, -1.246087, -2.653414, -0.812888, 1.570796, 1.718377],accel_mss,speed_ms,0,blend_radius_m)
    movel([0.147363, -1.247199, -2.652824, -0.812365, 1.570796, 1.718159],accel_mss,speed_ms,0,blend_radius_m)
    movel([0.147089, -1.248042, -2.652377, -0.811970, 1.570796, 1.717886],accel_mss,speed_ms,0,blend_radius_m)
    movel([0.145883, -1.250181, -2.651238, -0.810970, 1.570796, 1.716679],accel_mss,speed_ms,0,blend_radius_m)
    movel([0.144114, -1.252178, -2.650169, -0.810042, 1.570796, 1.714911],accel_mss,speed_ms,0,blend_radius_m)
    movel([0.142022, -1.253780, -2.649308, -0.809300, 1.570796, 1.712819],accel_mss,speed_ms,0,blend_radius_m)
    movel([0.139874, -1.254782, -2.648769, -0.808838, 1.570796, 1.710670],accel_mss,speed_ms,0,blend_radius_m)
    movel([0.139347, -1.254993, -2.648655, -0.808741, 1.570796, 1.710143],accel_mss,speed_ms,0,blend_radius_m)
    movel([0.139026, -1.255205, -2.648540, -0.808644, 1.570796, 1.709822],accel_mss,speed_ms,0,blend_radius_m)
    movel([0.138790, -1.255798, -2.648220, -0.808371, 1.570796, 1.709586],accel_mss,speed_ms,0,blend_radius_m)
    movel([0.138626, -1.256330, -2.647932, -0.808127, 1.570796, 1.709423],accel_mss,speed_ms,0,blend_radius_m)
    movel([0.138465, -1.256921, -2.647612, -0.807856, 1.570796, 1.709261],accel_mss,speed_ms,0,blend_radius_m)
    movel([0.138304, -1.257512, -2.647292, -0.807586, 1.570796, 1.709100],accel_mss,speed_ms,0,blend_radius_m)
    movel([0.138138, -1.258043, -2.647003, -0.807343, 1.570796, 1.708934],accel_mss,speed_ms,0,blend_radius_m)
    movel([0.137986, -1.258487, -2.646762, -0.807140, 1.570796, 1.708782],accel_mss,speed_ms,0,blend_radius_m)
    movel([0.137718, -1.258809, -2.646587, -0.806993, 1.570796, 1.708514],accel_mss,speed_ms,0,blend_radius_m)
    movel([0.137358, -1.258904, -2.646535, -0.806950, 1.570796, 1.708154],accel_mss,speed_ms,0,blend_radius_m)
    speed_ms = 0.003
    movel([0.137358, -1.262485, -2.648225, -0.801679, 1.570796, 1.708154],accel_mss,speed_ms,0,blend_radius_m)
    speed_ms = 0.007
    movel([0.137144, -1.262197, -2.648383, -0.801809, 1.570796, 1.707940],accel_mss,speed_ms,0,blend_radius_m)
    movel([0.137235, -1.261543, -2.648740, -0.802106, 1.570796, 1.708031],accel_mss,speed_ms,0,blend_radius_m)
    movel([0.137436, -1.260465, -2.649328, -0.802596, 1.570796, 1.708233],accel_mss,speed_ms,0,blend_radius_m)
    movel([0.137871, -1.258394, -2.650453, -0.803542, 1.570796, 1.708667],accel_mss,speed_ms,0,blend_radius_m)
    movel([0.138200, -1.256898, -2.651263, -0.804228, 1.570796, 1.708997],accel_mss,speed_ms,0,blend_radius_m)
    movel([0.138501, -1.255609, -2.651959, -0.804821, 1.570796, 1.709297],accel_mss,speed_ms,0,blend_radius_m)
    movel([0.138778, -1.254482, -2.652565, -0.805342, 1.570796, 1.709574],accel_mss,speed_ms,0,blend_radius_m)
    movel([0.139175, -1.254068, -2.652788, -0.805533, 1.570796, 1.709971],accel_mss,speed_ms,0,blend_radius_m)
    movel([0.139446, -1.253850, -2.652904, -0.805634, 1.570796, 1.710242],accel_mss,speed_ms,0,blend_radius_m)
    movel([0.139737, -1.253627, -2.653024, -0.805738, 1.570796, 1.710534],accel_mss,speed_ms,0,blend_radius_m)
    movel([0.140340, -1.253121, -2.653295, -0.805972, 1.570796, 1.711136],accel_mss,speed_ms,0,blend_radius_m)
    movel([0.140778, -1.252648, -2.653549, -0.806192, 1.570796, 1.711574],accel_mss,speed_ms,0,blend_radius_m)
    movel([0.141088, -1.252162, -2.653809, -0.806418, 1.570796, 1.711885],accel_mss,speed_ms,0,blend_radius_m)
    movel([0.141299, -1.251625, -2.654096, -0.806668, 1.570796, 1.712095],accel_mss,speed_ms,0,blend_radius_m)
    movel([0.141376, -1.251288, -2.654276, -0.806825, 1.570796, 1.712172],accel_mss,speed_ms,0,blend_radius_m)
    movel([0.141270, -1.250932, -2.654465, -0.806991, 1.570796, 1.712067],accel_mss,speed_ms,0,blend_radius_m)
    movel([0.141024, -1.250736, -2.654570, -0.807083, 1.570796, 1.711820],accel_mss,speed_ms,0,blend_radius_m)
    movel([0.140322, -1.250541, -2.654674, -0.807174, 1.570796, 1.711118],accel_mss,speed_ms,0,blend_radius_m)
    movel([0.139577, -1.250824, -2.654523, -0.807042, 1.570796, 1.710374],accel_mss,speed_ms,0,blend_radius_m)
    movel([0.138926, -1.251547, -2.654137, -0.806704, 1.570796, 1.709723],accel_mss,speed_ms,0,blend_radius_m)
    movel([0.138497, -1.252583, -2.653584, -0.806223, 1.570796, 1.709294],accel_mss,speed_ms,0,blend_radius_m)
    movel([0.138299, -1.253267, -2.653217, -0.805905, 1.570796, 1.709096],accel_mss,speed_ms,0,blend_radius_m)
    movel([0.138115, -1.253625, -2.653026, -0.805739, 1.570796, 1.708911],accel_mss,speed_ms,0,blend_radius_m)
    movel([0.137451, -1.254066, -2.652789, -0.805534, 1.570796, 1.708247],accel_mss,speed_ms,0,blend_radius_m)
    movel([0.137003, -1.254196, -2.652719, -0.805474, 1.570796, 1.707799],accel_mss,speed_ms,0,blend_radius_m)
    movel([0.136737, -1.254162, -2.652737, -0.805490, 1.570796, 1.707533],accel_mss,speed_ms,0,blend_radius_m)
    movel([0.136577, -1.253955, -2.652848, -0.805586, 1.570796, 1.707374],accel_mss,speed_ms,0,blend_radius_m)
    movel([0.136485, -1.253486, -2.653100, -0.805803, 1.570796, 1.707281],accel_mss,speed_ms,0,blend_radius_m)
    movel([0.136093, -1.252587, -2.653581, -0.806221, 1.570796, 1.706889],accel_mss,speed_ms,0,blend_radius_m)
    movel([0.135259, -1.252195, -2.653791, -0.806403, 1.570796, 1.706056],accel_mss,speed_ms,0,blend_radius_m)
    movel([0.134232, -1.252414, -2.653674, -0.806301, 1.570796, 1.705028],accel_mss,speed_ms,0,blend_radius_m)
    movel([0.133293, -1.253158, -2.653276, -0.805956, 1.570796, 1.704090],accel_mss,speed_ms,0,blend_radius_m)
    movel([0.132861, -1.253938, -2.652858, -0.805594, 1.570796, 1.703657],accel_mss,speed_ms,0,blend_radius_m)
    movel([0.132871, -1.254607, -2.652498, -0.805284, 1.570796, 1.703667],accel_mss,speed_ms,0,blend_radius_m)
    movel([0.133354, -1.255063, -2.652253, -0.805073, 1.570796, 1.704151],accel_mss,speed_ms,0,blend_radius_m)
    movel([0.134238, -1.255236, -2.652159, -0.804993, 1.570796, 1.705035],accel_mss,speed_ms,0,blend_radius_m)
    movel([0.134548, -1.255236, -2.652160, -0.804994, 1.570796, 1.705344],accel_mss,speed_ms,0,blend_radius_m)
    movel([0.134854, -1.255221, -2.652168, -0.805000, 1.570796, 1.705650],accel_mss,speed_ms,0,blend_radius_m)
    movel([0.135274, -1.255162, -2.652199, -0.805027, 1.570796, 1.706071],accel_mss,speed_ms,0,blend_radius_m)
    movel([0.135532, -1.255179, -2.652190, -0.805020, 1.570796, 1.706328],accel_mss,speed_ms,0,blend_radius_m)
    movel([0.135756, -1.255345, -2.652101, -0.804943, 1.570796, 1.706552],accel_mss,speed_ms,0,blend_radius_m)
    movel([0.135846, -1.255629, -2.651948, -0.804812, 1.570796, 1.706642],accel_mss,speed_ms,0,blend_radius_m)
    movel([0.135832, -1.256164, -2.651660, -0.804566, 1.570796, 1.706628],accel_mss,speed_ms,0,blend_radius_m)
    movel([0.135724, -1.257108, -2.651150, -0.804131, 1.570796, 1.706520],accel_mss,speed_ms,0,blend_radius_m)
    movel([0.135420, -1.259159, -2.650038, -0.803192, 1.570796, 1.706217],accel_mss,speed_ms,0,blend_radius_m)
    movel([0.135034, -1.261640, -2.648687, -0.802062, 1.570796, 1.705830],accel_mss,speed_ms,0,blend_radius_m)
    movel([0.134814, -1.262562, -2.648183, -0.801644, 1.570796, 1.705611],accel_mss,speed_ms,0,blend_radius_m)
    movel([0.134542, -1.263030, -2.647926, -0.801432, 1.570796, 1.705338],accel_mss,speed_ms,0,blend_radius_m)
    movel([0.134131, -1.263310, -2.647773, -0.801306, 1.570796, 1.704927],accel_mss,speed_ms,0,blend_radius_m)
    movel([0.133824, -1.263327, -2.647764, -0.801298, 1.570796, 1.704620],accel_mss,speed_ms,0,blend_radius_m)
    movel([0.133658, -1.263170, -2.647850, -0.801369, 1.570796, 1.704454],accel_mss,speed_ms,0,blend_radius_m)
    movel([0.133614, -1.262762, -2.648074, -0.801554, 1.570796, 1.704411],accel_mss,speed_ms,0,blend_radius_m)
    movel([0.133693, -1.261894, -2.648548, -0.801946, 1.570796, 1.704489],accel_mss,speed_ms,0,blend_radius_m)
    movel([0.133760, -1.261255, -2.648897, -0.802237, 1.570796, 1.704556],accel_mss,speed_ms,0,blend_radius_m)
    movel([0.133768, -1.260879, -2.649102, -0.802408, 1.570796, 1.704565],accel_mss,speed_ms,0,blend_radius_m)
    movel([0.133641, -1.260589, -2.649260, -0.802540, 1.570796, 1.704437],accel_mss,speed_ms,0,blend_radius_m)
    movel([0.133135, -1.260607, -2.649251, -0.802531, 1.570796, 1.703932],accel_mss,speed_ms,0,blend_radius_m)
    movel([0.132693, -1.260643, -2.649231, -0.802515, 1.570796, 1.703489],accel_mss,speed_ms,0,blend_radius_m)
    movel([0.132205, -1.260691, -2.649205, -0.802493, 1.570796, 1.703001],accel_mss,speed_ms,0,blend_radius_m)
    movel([0.131165, -1.260732, -2.649182, -0.802474, 1.570796, 1.701961],accel_mss,speed_ms,0,blend_radius_m)
    movel([0.130280, -1.260630, -2.649238, -0.802521, 1.570796, 1.701076],accel_mss,speed_ms,0,blend_radius_m)
    movel([0.129498, -1.260362, -2.649384, -0.802643, 1.570796, 1.700295],accel_mss,speed_ms,0,blend_radius_m)
    movel([0.128756, -1.259927, -2.649621, -0.802841, 1.570796, 1.699553],accel_mss,speed_ms,0,blend_radius_m)
    movel([0.127629, -1.258563, -2.650362, -0.803464, 1.570796, 1.698425],accel_mss,speed_ms,0,blend_radius_m)
    movel([0.127239, -1.256715, -2.651362, -0.804312, 1.570796, 1.698036],accel_mss,speed_ms,0,blend_radius_m)
    movel([0.127630, -1.254470, -2.652572, -0.805348, 1.570796, 1.698426],accel_mss,speed_ms,0,blend_radius_m)
    movel([0.128781, -1.251947, -2.653924, -0.806518, 1.570796, 1.699577],accel_mss,speed_ms,0,blend_radius_m)
    movel([0.129174, -1.251314, -2.654262, -0.806813, 1.570796, 1.699970],accel_mss,speed_ms,0,blend_radius_m)
    movel([0.129602, -1.250711, -2.654583, -0.807095, 1.570796, 1.700398],accel_mss,speed_ms,0,blend_radius_m)
    movel([0.130119, -1.250069, -2.654925, -0.807395, 1.570796, 1.700916],accel_mss,speed_ms,0,blend_radius_m)
    movel([0.130785, -1.249315, -2.655326, -0.807748, 1.570796, 1.701581],accel_mss,speed_ms,0,blend_radius_m)
    movel([0.132478, -1.247647, -2.656210, -0.808531, 1.570796, 1.703274],accel_mss,speed_ms,0,blend_radius_m)
    movel([0.134231, -1.246303, -2.656921, -0.809165, 1.570796, 1.705028],accel_mss,speed_ms,0,blend_radius_m)
    movel([0.136117, -1.245244, -2.657479, -0.809666, 1.570796, 1.706913],accel_mss,speed_ms,0,blend_radius_m)
    movel([0.138201, -1.244417, -2.657914, -0.810058, 1.570796, 1.708998],accel_mss,speed_ms,0,blend_radius_m)
    movel([0.139435, -1.244052, -2.658105, -0.810232, 1.570796, 1.710232],accel_mss,speed_ms,0,blend_radius_m)
    movel([0.140458, -1.243828, -2.658223, -0.810338, 1.570796, 1.711255],accel_mss,speed_ms,0,blend_radius_m)
    movel([0.141377, -1.243717, -2.658281, -0.810391, 1.570796, 1.712174],accel_mss,speed_ms,0,blend_radius_m)
    movel([0.142291, -1.243709, -2.658285, -0.810394, 1.570796, 1.713088],accel_mss,speed_ms,0,blend_radius_m)
    movel([0.144324, -1.244073, -2.658094, -0.810221, 1.570796, 1.715120],accel_mss,speed_ms,0,blend_radius_m)
    movel([0.145972, -1.244937, -2.657640, -0.809811, 1.570796, 1.716769],accel_mss,speed_ms,0,blend_radius_m)
    movel([0.147123, -1.246227, -2.656961, -0.809201, 1.570796, 1.717920],accel_mss,speed_ms,0,blend_radius_m)
    movel([0.147683, -1.247841, -2.656108, -0.808440, 1.570796, 1.718479],accel_mss,speed_ms,0,blend_radius_m)
    movel([0.147706, -1.248606, -2.655703, -0.808081, 1.570796, 1.718502],accel_mss,speed_ms,0,blend_radius_m)
